{attribute 'qualified_only'}
{attribute 'global_init_slot' := '50500'}
VAR_GLOBAL PERSISTENT
	//These tags are created here because you cannot write directly to local scoped tags(cpt_3144) from outside the POU
	//They are created here then mapped to the local variables in the POU
	//All tags in this GVL MUST have the {attribute 'OPC.UA.DA' :='1'} string above them in order to be exposed to OPC
	//Tags that are ONLY being read from the HMI have their values set in the opc_mapping program
	
		//------------------------------------------------------------------------------------------------------------------

	
	//State Mode
	{attribute 'OPC.UA.DA' :='1'}
	popa_0081_ed_routine_maint : BOOL;
	
//---HMI Commands--------------------------------------------------------------------------------------------------------------------------------------

	//Pumps-----------------------------------------------------------------------------------------------------------------------
	{attribute 'OPC.UA.DA' :='1'}
	popa_0081_u_3112_hmi_start_request: BOOL;
	{attribute 'OPC.UA.DA' :='1'}
	popa_0081_u_3212_hmi_start_request: BOOL;
	{attribute 'OPC.UA.DA' :='1'}
	popa_0081_u_3312_hmi_start_request: BOOL;
	{attribute 'OPC.UA.DA' :='1'}
	popa_0081_u_3160_hmi_start_request: BOOL;
	{attribute 'OPC.UA.DA' :='1'}
	popa_0081_u_3260_hmi_start_request: BOOL;
	{attribute 'OPC.UA.DA' :='1'}
	popa_0081_u_3360_hmi_start_request: BOOL;
	{attribute 'OPC.UA.DA' :='1'}
	popa_0081_u_3370_hmi_start_request: BOOL;
	{attribute 'OPC.UA.DA' :='1'}
	popa_0081_u_3405_hmi_start_request: BOOL;
		
	{attribute 'OPC.UA.DA' :='1'}
	popa_0081_u_3112_hmi_speed_request: REAL;
	{attribute 'OPC.UA.DA' :='1'}
	popa_0081_u_3212_hmi_speed_request: REAL;
	{attribute 'OPC.UA.DA' :='1'}
	popa_0081_u_3312_hmi_speed_request: REAL;
	{attribute 'OPC.UA.DA' :='1'}
	popa_0081_u_3160_hmi_speed_request: REAL;
	{attribute 'OPC.UA.DA' :='1'}
	popa_0081_u_3260_hmi_speed_request: REAL;
	{attribute 'OPC.UA.DA' :='1'}
	popa_0081_u_3360_hmi_speed_request: REAL;
	{attribute 'OPC.UA.DA' :='1'}
	popa_0081_u_3370_hmi_speed_request: REAL;
	{attribute 'OPC.UA.DA' :='1'}
	popa_0081_u_3405_hmi_speed_request: REAL;
	
	//Valves------------------------------------------------------------------------------------------------------------------------------
	{attribute 'OPC.UA.DA' :='1'}
	popa_0081_nv_3110_hmi_open_request: BOOL;
	{attribute 'OPC.UA.DA' :='1'}
	popa_0081_nv_3210_hmi_open_request: BOOL;
	{attribute 'OPC.UA.DA' :='1'}
	popa_0081_nv_3310_hmi_open_request: BOOL;
	{attribute 'OPC.UA.DA' :='1'}
	popa_0081_nv_3135_hmi_open_request: BOOL;
	{attribute 'OPC.UA.DA' :='1'}
	popa_0081_nv_3235_hmi_open_request: BOOL;
	{attribute 'OPC.UA.DA' :='1'}
	popa_0081_nv_3335_hmi_open_request: BOOL;
	{attribute 'OPC.UA.DA' :='1'}
	popa_0081_nv_3372_hmi_open_request: BOOL;
	{attribute 'OPC.UA.DA' :='1'}
	popa_0081_nv_3162_hmi_open_request: BOOL;
	
	//System date time year
	{attribute 'OPC.UA.DA' :='1'}
	popa_0081_system_date_time_year : INT;
	//System date time month
	{attribute 'OPC.UA.DA' :='1'}
	popa_0081_system_date_time_month : INT;
	//System date time day
	{attribute 'OPC.UA.DA' :='1'}
	popa_0081_system_date_time_day : INT;
	//System date time hour
	{attribute 'OPC.UA.DA' :='1'}
	popa_0081_system_date_time_hour : INT;
	//System date time minute
	{attribute 'OPC.UA.DA' :='1'}
	popa_0081_system_date_time_minute : INT;
	//System date time second
	{attribute 'OPC.UA.DA' :='1'}
	popa_0081_system_date_time_second : INT;
	//Hour setpoint for daily reset triggers
	{attribute 'OPC.UA.DA' :='1'}
	popa_0081_daily_reset_hour_setpoint : INT;
	//Minute setpoint for daily reset triggers
	{attribute 'OPC.UA.DA' :='1'}
	popa_0081_daily_reset_minute_setpoint : INT;
	//Alarm acknowledge, acks all alarms, clears lower priority level alarms
	{attribute 'OPC.UA.DA' :='1'}
	popa_0081_alarm_ack : BOOL;
	//Alarm reset, clears higher priority alarms
	{attribute 'OPC.UA.DA' :='1'}
	popa_0081_alarm_reset : BOOL;
	
	
	//------------------------------------------------------------------------------------------------------------------
	//Alarm Priority setpoint
	{attribute 'OPC.UA.DA' :='1'}
	popa_0081_av_3148_position_fail_priority : INT;
	//Alarm delay setpoint(seconds)
	{attribute 'OPC.UA.DA' :='1'}
	popa_0081_av_3148_position_fail_delay_setpoint : INT;
	//Alarm active for HMI
	{attribute 'OPC.UA.DA' :='1'}
	popa_0081_av_3148_position_fail_active : BOOL;
	//Alarm enable
	{attribute 'OPC.UA.DA' :='1'}
	popa_0081_av_3148_position_fail_enable: BOOL;
	//------------------------------------------------------------------------------------------------------------------
	//Alarm Priority setpoint
	{attribute 'OPC.UA.DA' :='1'}
	popa_0081_av_3248_position_fail_priority : INT;
	//Alarm delay setpoint(seconds)
	{attribute 'OPC.UA.DA' :='1'}
	popa_0081_av_3248_position_fail_delay_setpoint : INT;
	//Alarm active for HMI
	{attribute 'OPC.UA.DA' :='1'}
	popa_0081_av_3248_position_fail_active : BOOL;
	//Alarm enable
	{attribute 'OPC.UA.DA' :='1'}
	popa_0081_av_3248_position_fail_enable: BOOL;
	//------------------------------------------------------------------------------------------------------------------
	//Alarm Priority setpoint
	{attribute 'OPC.UA.DA' :='1'}
	popa_0081_av_3348_position_fail_priority : INT;
	//Alarm delay setpoint(seconds)
	{attribute 'OPC.UA.DA' :='1'}
	popa_0081_av_3348_position_fail_delay_setpoint : INT;
	//Alarm active for HMI
	{attribute 'OPC.UA.DA' :='1'}
	popa_0081_av_3348_position_fail_active : BOOL;
	//Alarm enable
	{attribute 'OPC.UA.DA' :='1'}
	popa_0081_av_3348_position_fail_enable: BOOL;
	
	//------------------------------------------------------------------------------------------------------------------
	//Alarm Priority setpoint
	{attribute 'OPC.UA.DA' :='1'}
	popa_0081_nv_3110_fail_to_open_priority : INT;
	//Alarm delay setpoint(seconds)
	{attribute 'OPC.UA.DA' :='1'}
	popa_0081_nv_3110_fail_to_open_delay_setpoint : INT;
	//Alarm active for HMI
	{attribute 'OPC.UA.DA' :='1'}
	popa_0081_nv_3110_fail_to_open_active : BOOL;
	//Alarm enable
	{attribute 'OPC.UA.DA' :='1'}
	popa_0081_nv_3110_fail_to_open_enable: BOOL;
	
	//Alarm Priority setpoint
	{attribute 'OPC.UA.DA' :='1'}
	popa_0081_nv_3110_fail_to_close_priority : INT;
	//Alarm delay setpoint(seconds)
	{attribute 'OPC.UA.DA' :='1'}
	popa_0081_nv_3110_fail_to_close_delay_setpoint : INT;
	//Alarm active for HMI
	{attribute 'OPC.UA.DA' :='1'}
	popa_0081_nv_3110_fail_to_close_active : BOOL;
	//Alarm enable
	{attribute 'OPC.UA.DA' :='1'}
	popa_0081_nv_3110_fail_to_close_enable: BOOL;
	
	//------------------------------------------------------------------------------------------------------------------
	//Alarm Priority setpoint
	{attribute 'OPC.UA.DA' :='1'}
	popa_0081_nv_3210_fail_to_open_priority : INT;
	//Alarm delay setpoint(seconds)
	{attribute 'OPC.UA.DA' :='1'}
	popa_0081_nv_3210_fail_to_open_delay_setpoint : INT;
	//Alarm active for HMI
	{attribute 'OPC.UA.DA' :='1'}
	popa_0081_nv_3210_fail_to_open_active : BOOL;
	//Alarm enable
	{attribute 'OPC.UA.DA' :='1'}
	popa_0081_nv_3210_fail_to_open_enable: BOOL;
	
	//Alarm Priority setpoint
	{attribute 'OPC.UA.DA' :='1'}
	popa_0081_nv_3210_fail_to_close_priority : INT;
	//Alarm delay setpoint(seconds)
	{attribute 'OPC.UA.DA' :='1'}
	popa_0081_nv_3210_fail_to_close_delay_setpoint : INT;
	//Alarm active for HMI
	{attribute 'OPC.UA.DA' :='1'}
	popa_0081_nv_3210_fail_to_close_active : BOOL;
	//Alarm enable
	{attribute 'OPC.UA.DA' :='1'}
	popa_0081_nv_3210_fail_to_close_enable: BOOL;
	
	//------------------------------------------------------------------------------------------------------------------
	//Alarm Priority setpoint
	{attribute 'OPC.UA.DA' :='1'}
	popa_0081_nv_3310_fail_to_open_priority : INT;
	//Alarm delay setpoint(seconds)
	{attribute 'OPC.UA.DA' :='1'}
	popa_0081_nv_3310_fail_to_open_delay_setpoint : INT;
	//Alarm active for HMI
	{attribute 'OPC.UA.DA' :='1'}
	popa_0081_nv_3310_fail_to_open_active : BOOL;
	//Alarm enable
	{attribute 'OPC.UA.DA' :='1'}
	popa_0081_nv_3310_fail_to_open_enable: BOOL;
	
	//Alarm Priority setpoint
	{attribute 'OPC.UA.DA' :='1'}
	popa_0081_nv_3310_fail_to_close_priority : INT;
	//Alarm delay setpoint(seconds)
	{attribute 'OPC.UA.DA' :='1'}
	popa_0081_nv_3310_fail_to_close_delay_setpoint : INT;
	//Alarm active for HMI
	{attribute 'OPC.UA.DA' :='1'}
	popa_0081_nv_3310_fail_to_close_active : BOOL;
	//Alarm enable
	{attribute 'OPC.UA.DA' :='1'}
	popa_0081_nv_3310_fail_to_close_enable: BOOL;
	
	//------------------------------------------------------------------------------------------------------------------
	//Alarm Priority setpoint
	{attribute 'OPC.UA.DA' :='1'}
	popa_0081_nv_3135_fail_to_open_priority : INT;
	//Alarm delay setpoint(seconds)
	{attribute 'OPC.UA.DA' :='1'}
	popa_0081_nv_3135_fail_to_open_delay_setpoint : INT;
	//Alarm active for HMI
	{attribute 'OPC.UA.DA' :='1'}
	popa_0081_nv_3135_fail_to_open_active : BOOL;
	//Alarm enable
	{attribute 'OPC.UA.DA' :='1'}
	popa_0081_nv_3135_fail_to_open_enable: BOOL;
	
	//Alarm Priority setpoint
	{attribute 'OPC.UA.DA' :='1'}
	popa_0081_nv_3135_fail_to_close_priority : INT;
	//Alarm delay setpoint(seconds)
	{attribute 'OPC.UA.DA' :='1'}
	popa_0081_nv_3135_fail_to_close_delay_setpoint : INT;
	//Alarm active for HMI
	{attribute 'OPC.UA.DA' :='1'}
	popa_0081_nv_3135_fail_to_close_active : BOOL;
	//Alarm enable
	{attribute 'OPC.UA.DA' :='1'}
	popa_0081_nv_3135_fail_to_close_enable: BOOL;
	
	//------------------------------------------------------------------------------------------------------------------
	//Alarm Priority setpoint
	{attribute 'OPC.UA.DA' :='1'}
	popa_0081_nv_3235_fail_to_open_priority : INT;
	//Alarm delay setpoint(seconds)
	{attribute 'OPC.UA.DA' :='1'}
	popa_0081_nv_3235_fail_to_open_delay_setpoint : INT;
	//Alarm active for HMI
	{attribute 'OPC.UA.DA' :='1'}
	popa_0081_nv_3235_fail_to_open_active : BOOL;
	//Alarm enable
	{attribute 'OPC.UA.DA' :='1'}
	popa_0081_nv_3235_fail_to_open_enable: BOOL;
	
	//Alarm Priority setpoint
	{attribute 'OPC.UA.DA' :='1'}
	popa_0081_nv_3235_fail_to_close_priority : INT;
	//Alarm delay setpoint(seconds)
	{attribute 'OPC.UA.DA' :='1'}
	popa_0081_nv_3235_fail_to_close_delay_setpoint : INT;
	//Alarm active for HMI
	{attribute 'OPC.UA.DA' :='1'}
	popa_0081_nv_3235_fail_to_close_active : BOOL;
	//Alarm enable
	{attribute 'OPC.UA.DA' :='1'}
	popa_0081_nv_3235_fail_to_close_enable: BOOL;
	
	//------------------------------------------------------------------------------------------------------------------
	//Alarm Priority setpoint
	{attribute 'OPC.UA.DA' :='1'}
	popa_0081_nv_3335_fail_to_open_priority : INT;
	//Alarm delay setpoint(seconds)
	{attribute 'OPC.UA.DA' :='1'}
	popa_0081_nv_3335_fail_to_open_delay_setpoint : INT;
	//Alarm active for HMI
	{attribute 'OPC.UA.DA' :='1'}
	popa_0081_nv_3335_fail_to_open_active : BOOL;
	//Alarm enable
	{attribute 'OPC.UA.DA' :='1'}
	popa_0081_nv_3335_fail_to_open_enable: BOOL;
	
	//Alarm Priority setpoint
	{attribute 'OPC.UA.DA' :='1'}
	popa_0081_nv_3335_fail_to_close_priority : INT;
	//Alarm delay setpoint(seconds)
	{attribute 'OPC.UA.DA' :='1'}
	popa_0081_nv_3335_fail_to_close_delay_setpoint : INT;
	//Alarm active for HMI
	{attribute 'OPC.UA.DA' :='1'}
	popa_0081_nv_3335_fail_to_close_active : BOOL;
	//Alarm enable
	{attribute 'OPC.UA.DA' :='1'}
	popa_0081_nv_3335_fail_to_close_enable: BOOL;
	
	//------------------------------------------------------------------------------------------------------------------
	//Alarm Priority setpoint
	{attribute 'OPC.UA.DA' :='1'}
	popa_0081_nv_3372_fail_to_open_priority : INT;
	//Alarm delay setpoint(seconds)
	{attribute 'OPC.UA.DA' :='1'}
	popa_0081_nv_3372_fail_to_open_delay_setpoint : INT;
	//Alarm active for HMI
	{attribute 'OPC.UA.DA' :='1'}
	popa_0081_nv_3372_fail_to_open_active : BOOL;
	//Alarm enable
	{attribute 'OPC.UA.DA' :='1'}
	popa_0081_nv_3372_fail_to_open_enable: BOOL;
	
	//Alarm Priority setpoint
	{attribute 'OPC.UA.DA' :='1'}
	popa_0081_nv_3372_fail_to_close_priority : INT;
	//Alarm delay setpoint(seconds)
	{attribute 'OPC.UA.DA' :='1'}
	popa_0081_nv_3372_fail_to_close_delay_setpoint : INT;
	//Alarm active for HMI
	{attribute 'OPC.UA.DA' :='1'}
	popa_0081_nv_3372_fail_to_close_active : BOOL;
	//Alarm enable
	{attribute 'OPC.UA.DA' :='1'}
	popa_0081_nv_3372_fail_to_close_enable: BOOL;
	
	//------------------------------------------------------------------------------------------------------------------
	//Alarm Priority setpoint
	{attribute 'OPC.UA.DA' :='1'}
	popa_0081_nv_3162_fail_to_open_priority : INT;
	//Alarm delay setpoint(seconds)
	{attribute 'OPC.UA.DA' :='1'}
	popa_0081_nv_3162_fail_to_open_delay_setpoint : INT;
	//Alarm active for HMI
	{attribute 'OPC.UA.DA' :='1'}
	popa_0081_nv_3162_fail_to_open_active : BOOL;
	//Alarm enable
	{attribute 'OPC.UA.DA' :='1'}
	popa_0081_nv_3162_fail_to_open_enable: BOOL;
	
	//Alarm Priority setpoint
	{attribute 'OPC.UA.DA' :='1'}
	popa_0081_nv_3162_fail_to_close_priority : INT;
	//Alarm delay setpoint(seconds)
	{attribute 'OPC.UA.DA' :='1'}
	popa_0081_nv_3162_fail_to_close_delay_setpoint : INT;
	//Alarm active for HMI
	{attribute 'OPC.UA.DA' :='1'}
	popa_0081_nv_3162_fail_to_close_active : BOOL;
	//Alarm enable
	{attribute 'OPC.UA.DA' :='1'}
	popa_0081_nv_3162_fail_to_close_enable: BOOL;
	


//---Pumps-------------------------------------------------------------------------------------------------------------------------------------
	//------------------------------------------------------------------------------------------------------------------
	//Alarm Priority setpoint
	{attribute 'OPC.UA.DA' :='1'}
	popa_0081_u_3112_fail_to_start_priority : INT;
	//Alarm delay setpoint(seconds)
	{attribute 'OPC.UA.DA' :='1'}
	popa_0081_u_3112_fail_to_start_delay_setpoint : INT;
	//Alarm active for HMI
	{attribute 'OPC.UA.DA' :='1'}
	popa_0081_u_3112_fail_to_start_active : BOOL;
	//Alarm enable
	{attribute 'OPC.UA.DA' :='1'}
	popa_0081_u_3112_fail_to_start_enable: BOOL;
	
	//Alarm Priority setpoint
	{attribute 'OPC.UA.DA' :='1'}
	popa_0081_u_3112_fail_to_stop_priority : INT;
	//Alarm delay setpoint(seconds)
	{attribute 'OPC.UA.DA' :='1'}
	popa_0081_u_3112_fail_to_stop_delay_setpoint : INT;
	//Alarm active for HMI
	{attribute 'OPC.UA.DA' :='1'}
	popa_0081_u_3112_fail_to_stop_active : BOOL;
	//Alarm enable
	{attribute 'OPC.UA.DA' :='1'}
	popa_0081_u_3112_fail_to_stop_enable: BOOL;
	
	//------------------------------------------------------------------------------------------------------------------
	//Alarm Priority setpoint
	{attribute 'OPC.UA.DA' :='1'}
	popa_0081_u_3212_fail_to_start_priority : INT;
	//Alarm delay setpoint(seconds)
	{attribute 'OPC.UA.DA' :='1'}
	popa_0081_u_3212_fail_to_start_delay_setpoint : INT;
	//Alarm active for HMI
	{attribute 'OPC.UA.DA' :='1'}
	popa_0081_u_3212_fail_to_start_active : BOOL;
	//Alarm enable
	{attribute 'OPC.UA.DA' :='1'}
	popa_0081_u_3212_fail_to_start_enable: BOOL;
	
	//Alarm Priority setpoint
	{attribute 'OPC.UA.DA' :='1'}
	popa_0081_u_3212_fail_to_stop_priority : INT;
	//Alarm delay setpoint(seconds)
	{attribute 'OPC.UA.DA' :='1'}
	popa_0081_u_3212_fail_to_stop_delay_setpoint : INT;
	//Alarm active for HMI
	{attribute 'OPC.UA.DA' :='1'}
	popa_0081_u_3212_fail_to_stop_active : BOOL;
	//Alarm enable
	{attribute 'OPC.UA.DA' :='1'}
	popa_0081_u_3212_fail_to_stop_enable: BOOL;
	
	//------------------------------------------------------------------------------------------------------------------
	//Alarm Priority setpoint
	{attribute 'OPC.UA.DA' :='1'}
	popa_0081_u_3312_fail_to_start_priority : INT;
	//Alarm delay setpoint(seconds)
	{attribute 'OPC.UA.DA' :='1'}
	popa_0081_u_3312_fail_to_start_delay_setpoint : INT;
	//Alarm active for HMI
	{attribute 'OPC.UA.DA' :='1'}
	popa_0081_u_3312_fail_to_start_active : BOOL;
	//Alarm enable
	{attribute 'OPC.UA.DA' :='1'}
	popa_0081_u_3312_fail_to_start_enable: BOOL;
	
	//Alarm Priority setpoint
	{attribute 'OPC.UA.DA' :='1'}
	popa_0081_u_3312_fail_to_stop_priority : INT;
	//Alarm delay setpoint(seconds)
	{attribute 'OPC.UA.DA' :='1'}
	popa_0081_u_3312_fail_to_stop_delay_setpoint : INT;
	//Alarm active for HMI
	{attribute 'OPC.UA.DA' :='1'}
	popa_0081_u_3312_fail_to_stop_active : BOOL;
	//Alarm enable
	{attribute 'OPC.UA.DA' :='1'}
	popa_0081_u_3312_fail_to_stop_enable: BOOL;
	
	//------------------------------------------------------------------------------------------------------------------
	//Alarm Priority setpoint
	{attribute 'OPC.UA.DA' :='1'}
	popa_0081_u_3160_fail_to_start_priority : INT;
	//Alarm delay setpoint(seconds)
	{attribute 'OPC.UA.DA' :='1'}
	popa_0081_u_3160_fail_to_start_delay_setpoint : INT;
	//Alarm active for HMI
	{attribute 'OPC.UA.DA' :='1'}
	popa_0081_u_3160_fail_to_start_active : BOOL;
	//Alarm enable
	{attribute 'OPC.UA.DA' :='1'}
	popa_0081_u_3160_fail_to_start_enable: BOOL;
	
	//Alarm Priority setpoint
	{attribute 'OPC.UA.DA' :='1'}
	popa_0081_u_3160_fail_to_stop_priority : INT;
	//Alarm delay setpoint(seconds)
	{attribute 'OPC.UA.DA' :='1'}
	popa_0081_u_3160_fail_to_stop_delay_setpoint : INT;
	//Alarm active for HMI
	{attribute 'OPC.UA.DA' :='1'}
	popa_0081_u_3160_fail_to_stop_active : BOOL;
	//Alarm enable
	{attribute 'OPC.UA.DA' :='1'}
	popa_0081_u_3160_fail_to_stop_enable: BOOL;
	
	//------------------------------------------------------------------------------------------------------------------
	//Alarm Priority setpoint
	{attribute 'OPC.UA.DA' :='1'}
	popa_0081_u_3260_fail_to_start_priority : INT;
	//Alarm delay setpoint(seconds)
	{attribute 'OPC.UA.DA' :='1'}
	popa_0081_u_3260_fail_to_start_delay_setpoint : INT;
	//Alarm active for HMI
	{attribute 'OPC.UA.DA' :='1'}
	popa_0081_u_3260_fail_to_start_active : BOOL;
	//Alarm enable
	{attribute 'OPC.UA.DA' :='1'}
	popa_0081_u_3260_fail_to_start_enable: BOOL;
	
	//Alarm Priority setpoint
	{attribute 'OPC.UA.DA' :='1'}
	popa_0081_u_3260_fail_to_stop_priority : INT;
	//Alarm delay setpoint(seconds)
	{attribute 'OPC.UA.DA' :='1'}
	popa_0081_u_3260_fail_to_stop_delay_setpoint : INT;
	//Alarm active for HMI
	{attribute 'OPC.UA.DA' :='1'}
	popa_0081_u_3260_fail_to_stop_active : BOOL;
	//Alarm enable
	{attribute 'OPC.UA.DA' :='1'}
	popa_0081_u_3260_fail_to_stop_enable: BOOL;
	
	//------------------------------------------------------------------------------------------------------------------
	//Alarm Priority setpoint
	{attribute 'OPC.UA.DA' :='1'}
	popa_0081_u_3360_fail_to_start_priority : INT;
	//Alarm delay setpoint(seconds)
	{attribute 'OPC.UA.DA' :='1'}
	popa_0081_u_3360_fail_to_start_delay_setpoint : INT;
	//Alarm active for HMI
	{attribute 'OPC.UA.DA' :='1'}
	popa_0081_u_3360_fail_to_start_active : BOOL;
	//Alarm enable
	{attribute 'OPC.UA.DA' :='1'}
	popa_0081_u_3360_fail_to_start_enable: BOOL;
	
	//Alarm Priority setpoint
	{attribute 'OPC.UA.DA' :='1'}
	popa_0081_u_3360_fail_to_stop_priority : INT;
	//Alarm delay setpoint(seconds)
	{attribute 'OPC.UA.DA' :='1'}
	popa_0081_u_3360_fail_to_stop_delay_setpoint : INT;
	//Alarm active for HMI
	{attribute 'OPC.UA.DA' :='1'}
	popa_0081_u_3360_fail_to_stop_active : BOOL;
	//Alarm enable
	{attribute 'OPC.UA.DA' :='1'}
	popa_0081_u_3360_fail_to_stop_enable: BOOL;
	
	//------------------------------------------------------------------------------------------------------------------
	//Alarm Priority setpoint
	{attribute 'OPC.UA.DA' :='1'}
	popa_0081_u_3370_fail_to_start_priority : INT;
	//Alarm delay setpoint(seconds)
	{attribute 'OPC.UA.DA' :='1'}
	popa_0081_u_3370_fail_to_start_delay_setpoint : INT;
	//Alarm active for HMI
	{attribute 'OPC.UA.DA' :='1'}
	popa_0081_u_3370_fail_to_start_active : BOOL;
	//Alarm enable
	{attribute 'OPC.UA.DA' :='1'}
	popa_0081_u_3370_fail_to_start_enable: BOOL;
	
	//Alarm Priority setpoint
	{attribute 'OPC.UA.DA' :='1'}
	popa_0081_u_3370_fail_to_stop_priority : INT;
	//Alarm delay setpoint(seconds)
	{attribute 'OPC.UA.DA' :='1'}
	popa_0081_u_3370_fail_to_stop_delay_setpoint : INT;
	//Alarm active for HMI
	{attribute 'OPC.UA.DA' :='1'}
	popa_0081_u_3370_fail_to_stop_active : BOOL;
	//Alarm enable
	{attribute 'OPC.UA.DA' :='1'}
	popa_0081_u_3370_fail_to_stop_enable: BOOL;
	
	//------------------------------------------------------------------------------------------------------------------
	//Alarm Priority setpoint
	{attribute 'OPC.UA.DA' :='1'}
	popa_0081_u_3405_fail_to_start_priority : INT;
	//Alarm delay setpoint(seconds)
	{attribute 'OPC.UA.DA' :='1'}
	popa_0081_u_3405_fail_to_start_delay_setpoint : INT;
	//Alarm active for HMI
	{attribute 'OPC.UA.DA' :='1'}
	popa_0081_u_3405_fail_to_start_active : BOOL;
	//Alarm enable
	{attribute 'OPC.UA.DA' :='1'}
	popa_0081_u_3405_fail_to_start_enable: BOOL;
	
	//Alarm Priority setpoint
	{attribute 'OPC.UA.DA' :='1'}
	popa_0081_u_3405_fail_to_stop_priority : INT;
	//Alarm delay setpoint(seconds)
	{attribute 'OPC.UA.DA' :='1'}
	popa_0081_u_3405_fail_to_stop_delay_setpoint : INT;
	//Alarm active for HMI
	{attribute 'OPC.UA.DA' :='1'}
	popa_0081_u_3405_fail_to_stop_active : BOOL;
	//Alarm enable
	{attribute 'OPC.UA.DA' :='1'}
	popa_0081_u_3405_fail_to_stop_enable: BOOL;

	
	//---------------------------------------------------------------------------------------------------------
	//Raw Min value for analog input
	{attribute 'OPC.UA.DA' :='1'}
	popa_0081_u_3112_speed_command_raw_min : REAL :=0;
	//Raw max value for analog input
	{attribute 'OPC.UA.DA' :='1'}
	popa_0081_u_3112_speed_command_raw_max : REAL :=32767;
	//EU Min value for analog input
	{attribute 'OPC.UA.DA' :='1'}
	popa_0081_u_3112_speed_command_eu_min : REAL;
	//EU Max value for analog input
	{attribute 'OPC.UA.DA' :='1'}
	popa_0081_u_3112_speed_command_eu_max : REAL;
	//Filter factor value for analog input
	{attribute 'OPC.UA.DA' :='1'}
	popa_0081_u_3112_speed_command_filter_factor : REAL;
	//Scaled value for analog input
	{attribute 'OPC.UA.DA' :='1'}
	popa_0081_u_3112_speed_command_scaled_value : REAL;
	
	//Raw Min value for analog input
	{attribute 'OPC.UA.DA' :='1'}
	popa_0081_u_3112_speed_feedback_raw_min : REAL :=0;
	//Raw max value for analog input
	{attribute 'OPC.UA.DA' :='1'}
	popa_0081_u_3112_speed_feedback_raw_max : REAL :=32767;
	//EU Min value for analog input
	{attribute 'OPC.UA.DA' :='1'}
	popa_0081_u_3112_speed_feedback_eu_min : REAL;
	//EU Max value for analog input
	{attribute 'OPC.UA.DA' :='1'}
	popa_0081_u_3112_speed_feedback_eu_max : REAL;
	//Filter factor value for analog input
	{attribute 'OPC.UA.DA' :='1'}
	popa_0081_u_3112_speed_feedback_filter_factor : REAL;
	//Scaled value for analog input
	{attribute 'OPC.UA.DA' :='1'}
	popa_0081_u_3112_speed_feedback_scaled_value : REAL;
	
	
	//---------------------------------------------------------------------------------------------------------
	//Raw Min value for analog input
	{attribute 'OPC.UA.DA' :='1'}
	popa_0081_u_3212_speed_command_raw_min : REAL :=0;
	//Raw max value for analog input
	{attribute 'OPC.UA.DA' :='1'}
	popa_0081_u_3212_speed_command_raw_max : REAL :=32767;
	//EU Min value for analog input
	{attribute 'OPC.UA.DA' :='1'}
	popa_0081_u_3212_speed_command_eu_min : REAL;
	//EU Max value for analog input
	{attribute 'OPC.UA.DA' :='1'}
	popa_0081_u_3212_speed_command_eu_max : REAL;
	//Filter factor value for analog input
	{attribute 'OPC.UA.DA' :='1'}
	popa_0081_u_3212_speed_command_filter_factor : REAL;
	//Scaled value for analog input
	{attribute 'OPC.UA.DA' :='1'}
	popa_0081_u_3212_speed_command_scaled_value : REAL;
	
	//Raw Min value for analog input
	{attribute 'OPC.UA.DA' :='1'}
	popa_0081_u_3212_speed_feedback_raw_min : REAL :=0;
	//Raw max value for analog input
	{attribute 'OPC.UA.DA' :='1'}
	popa_0081_u_3212_speed_feedback_raw_max : REAL :=32767;
	//EU Min value for analog input
	{attribute 'OPC.UA.DA' :='1'}
	popa_0081_u_3212_speed_feedback_eu_min : REAL;
	//EU Max value for analog input
	{attribute 'OPC.UA.DA' :='1'}
	popa_0081_u_3212_speed_feedback_eu_max : REAL;
	//Filter factor value for analog input
	{attribute 'OPC.UA.DA' :='1'}
	popa_0081_u_3212_speed_feedback_filter_factor : REAL;
	//Scaled value for analog input
	{attribute 'OPC.UA.DA' :='1'}
	popa_0081_u_3212_speed_feedback_scaled_value : REAL;
	
	
	//---------------------------------------------------------------------------------------------------------
	//Raw Min value for analog input
	{attribute 'OPC.UA.DA' :='1'}
	popa_0081_u_3312_speed_command_raw_min : REAL :=0;
	//Raw max value for analog input
	{attribute 'OPC.UA.DA' :='1'}
	popa_0081_u_3312_speed_command_raw_max : REAL :=32767;
	//EU Min value for analog input
	{attribute 'OPC.UA.DA' :='1'}
	popa_0081_u_3312_speed_command_eu_min : REAL;
	//EU Max value for analog input
	{attribute 'OPC.UA.DA' :='1'}
	popa_0081_u_3312_speed_command_eu_max : REAL;
	//Filter factor value for analog input
	{attribute 'OPC.UA.DA' :='1'}
	popa_0081_u_3312_speed_command_filter_factor : REAL;
	//Scaled value for analog input
	{attribute 'OPC.UA.DA' :='1'}
	popa_0081_u_3312_speed_command_scaled_value : REAL;
	
	//Raw Min value for analog input
	{attribute 'OPC.UA.DA' :='1'}
	popa_0081_u_3312_speed_feedback_raw_min : REAL :=0;
	//Raw max value for analog input
	{attribute 'OPC.UA.DA' :='1'}
	popa_0081_u_3312_speed_feedback_raw_max : REAL :=32767;
	//EU Min value for analog input
	{attribute 'OPC.UA.DA' :='1'}
	popa_0081_u_3312_speed_feedback_eu_min : REAL;
	//EU Max value for analog input
	{attribute 'OPC.UA.DA' :='1'}
	popa_0081_u_3312_speed_feedback_eu_max : REAL;
	//Filter factor value for analog input
	{attribute 'OPC.UA.DA' :='1'}
	popa_0081_u_3312_speed_feedback_filter_factor : REAL;
	//Scaled value for analog input
	{attribute 'OPC.UA.DA' :='1'}
	popa_0081_u_3312_speed_feedback_scaled_value : REAL;
	
	
	//---------------------------------------------------------------------------------------------------------
	//Raw Min value for analog input
	{attribute 'OPC.UA.DA' :='1'}
	popa_0081_u_3160_speed_command_raw_min : REAL :=0;
	//Raw max value for analog input
	{attribute 'OPC.UA.DA' :='1'}
	popa_0081_u_3160_speed_command_raw_max : REAL :=32767;
	//EU Min value for analog input
	{attribute 'OPC.UA.DA' :='1'}
	popa_0081_u_3160_speed_command_eu_min : REAL;
	//EU Max value for analog input
	{attribute 'OPC.UA.DA' :='1'}
	popa_0081_u_3160_speed_command_eu_max : REAL;
	//Filter factor value for analog input
	{attribute 'OPC.UA.DA' :='1'}
	popa_0081_u_3160_speed_command_filter_factor : REAL;
	//Scaled value for analog input
	{attribute 'OPC.UA.DA' :='1'}
	popa_0081_u_3160_speed_command_scaled_value : REAL;
	
	//Raw Min value for analog input
	{attribute 'OPC.UA.DA' :='1'}
	popa_0081_u_3160_speed_feedback_raw_min : REAL :=0;
	//Raw max value for analog input
	{attribute 'OPC.UA.DA' :='1'}
	popa_0081_u_3160_speed_feedback_raw_max : REAL :=32767;
	//EU Min value for analog input
	{attribute 'OPC.UA.DA' :='1'}
	popa_0081_u_3160_speed_feedback_eu_min : REAL;
	//EU Max value for analog input
	{attribute 'OPC.UA.DA' :='1'}
	popa_0081_u_3160_speed_feedback_eu_max : REAL;
	//Filter factor value for analog input
	{attribute 'OPC.UA.DA' :='1'}
	popa_0081_u_3160_speed_feedback_filter_factor : REAL;
	//Scaled value for analog input
	{attribute 'OPC.UA.DA' :='1'}
	popa_0081_u_3160_speed_feedback_scaled_value : REAL;
	
	
	//---------------------------------------------------------------------------------------------------------
	//Raw Min value for analog input
	{attribute 'OPC.UA.DA' :='1'}
	popa_0081_u_3260_speed_command_raw_min : REAL :=0;
	//Raw max value for analog input
	{attribute 'OPC.UA.DA' :='1'}
	popa_0081_u_3260_speed_command_raw_max : REAL :=32767;
	//EU Min value for analog input
	{attribute 'OPC.UA.DA' :='1'}
	popa_0081_u_3260_speed_command_eu_min : REAL;
	//EU Max value for analog input
	{attribute 'OPC.UA.DA' :='1'}
	popa_0081_u_3260_speed_command_eu_max : REAL;
	//Filter factor value for analog input
	{attribute 'OPC.UA.DA' :='1'}
	popa_0081_u_3260_speed_command_filter_factor : REAL;
	//Scaled value for analog input
	{attribute 'OPC.UA.DA' :='1'}
	popa_0081_u_3260_speed_command_scaled_value : REAL;
	
	//Raw Min value for analog input
	{attribute 'OPC.UA.DA' :='1'}
	popa_0081_u_3260_speed_feedback_raw_min : REAL :=0;
	//Raw max value for analog input
	{attribute 'OPC.UA.DA' :='1'}
	popa_0081_u_3260_speed_feedback_raw_max : REAL :=32767;
	//EU Min value for analog input
	{attribute 'OPC.UA.DA' :='1'}
	popa_0081_u_3260_speed_feedback_eu_min : REAL;
	//EU Max value for analog input
	{attribute 'OPC.UA.DA' :='1'}
	popa_0081_u_3260_speed_feedback_eu_max : REAL;
	//Filter factor value for analog input
	{attribute 'OPC.UA.DA' :='1'}
	popa_0081_u_3260_speed_feedback_filter_factor : REAL;
	//Scaled value for analog input
	{attribute 'OPC.UA.DA' :='1'}
	popa_0081_u_3260_speed_feedback_scaled_value : REAL;
	
	
	//---------------------------------------------------------------------------------------------------------
	//Raw Min value for analog input
	{attribute 'OPC.UA.DA' :='1'}
	popa_0081_u_3360_speed_command_raw_min : REAL :=0;
	//Raw max value for analog input
	{attribute 'OPC.UA.DA' :='1'}
	popa_0081_u_3360_speed_command_raw_max : REAL :=32767;
	//EU Min value for analog input
	{attribute 'OPC.UA.DA' :='1'}
	popa_0081_u_3360_speed_command_eu_min : REAL;
	//EU Max value for analog input
	{attribute 'OPC.UA.DA' :='1'}
	popa_0081_u_3360_speed_command_eu_max : REAL;
	//Filter factor value for analog input
	{attribute 'OPC.UA.DA' :='1'}
	popa_0081_u_3360_speed_command_filter_factor : REAL;
	//Scaled value for analog input
	{attribute 'OPC.UA.DA' :='1'}
	popa_0081_u_3360_speed_command_scaled_value : REAL;
	
	//Raw Min value for analog input
	{attribute 'OPC.UA.DA' :='1'}
	popa_0081_u_3360_speed_feedback_raw_min : REAL :=0;
	//Raw max value for analog input
	{attribute 'OPC.UA.DA' :='1'}
	popa_0081_u_3360_speed_feedback_raw_max : REAL :=32767;
	//EU Min value for analog input
	{attribute 'OPC.UA.DA' :='1'}
	popa_0081_u_3360_speed_feedback_eu_min : REAL;
	//EU Max value for analog input
	{attribute 'OPC.UA.DA' :='1'}
	popa_0081_u_3360_speed_feedback_eu_max : REAL;
	//Filter factor value for analog input
	{attribute 'OPC.UA.DA' :='1'}
	popa_0081_u_3360_speed_feedback_filter_factor : REAL;
	//Scaled value for analog input
	{attribute 'OPC.UA.DA' :='1'}
	popa_0081_u_3360_speed_feedback_scaled_value : REAL;
	
	
	//---------------------------------------------------------------------------------------------------------
	//Raw Min value for analog input
	{attribute 'OPC.UA.DA' :='1'}
	popa_0081_u_3370_speed_command_raw_min : REAL :=0;
	//Raw max value for analog input
	{attribute 'OPC.UA.DA' :='1'}
	popa_0081_u_3370_speed_command_raw_max : REAL :=32767;
	//EU Min value for analog input
	{attribute 'OPC.UA.DA' :='1'}
	popa_0081_u_3370_speed_command_eu_min : REAL;
	//EU Max value for analog input
	{attribute 'OPC.UA.DA' :='1'}
	popa_0081_u_3370_speed_command_eu_max : REAL;
	//Filter factor value for analog input
	{attribute 'OPC.UA.DA' :='1'}
	popa_0081_u_3370_speed_command_filter_factor : REAL;
	//Scaled value for analog input
	{attribute 'OPC.UA.DA' :='1'}
	popa_0081_u_3370_speed_command_scaled_value : REAL;
	
	//Raw Min value for analog input
	{attribute 'OPC.UA.DA' :='1'}
	popa_0081_u_3370_speed_feedback_raw_min : REAL :=0;
	//Raw max value for analog input
	{attribute 'OPC.UA.DA' :='1'}
	popa_0081_u_3370_speed_feedback_raw_max : REAL :=32767;
	//EU Min value for analog input
	{attribute 'OPC.UA.DA' :='1'}
	popa_0081_u_3370_speed_feedback_eu_min : REAL;
	//EU Max value for analog input
	{attribute 'OPC.UA.DA' :='1'}
	popa_0081_u_3370_speed_feedback_eu_max : REAL;
	//Filter factor value for analog input
	{attribute 'OPC.UA.DA' :='1'}
	popa_0081_u_3370_speed_feedback_filter_factor : REAL;
	//Scaled value for analog input
	{attribute 'OPC.UA.DA' :='1'}
	popa_0081_u_3370_speed_feedback_scaled_value : REAL;
	
	
	//---------------------------------------------------------------------------------------------------------
	//Raw Min value for analog input
	{attribute 'OPC.UA.DA' :='1'}
	popa_0081_u_3405_speed_command_raw_min : REAL :=0;
	//Raw max value for analog input
	{attribute 'OPC.UA.DA' :='1'}
	popa_0081_u_3405_speed_command_raw_max : REAL :=32767;
	//EU Min value for analog input
	{attribute 'OPC.UA.DA' :='1'}
	popa_0081_u_3405_speed_command_eu_min : REAL;
	//EU Max value for analog input
	{attribute 'OPC.UA.DA' :='1'}
	popa_0081_u_3405_speed_command_eu_max : REAL;
	//Filter factor value for analog input
	{attribute 'OPC.UA.DA' :='1'}
	popa_0081_u_3405_speed_command_filter_factor : REAL;
	//Scaled value for analog input
	{attribute 'OPC.UA.DA' :='1'}
	popa_0081_u_3405_speed_command_scaled_value : REAL;
	
	//Raw Min value for analog input
	{attribute 'OPC.UA.DA' :='1'}
	popa_0081_u_3405_speed_feedback_raw_min : REAL :=0;
	//Raw max value for analog input
	{attribute 'OPC.UA.DA' :='1'}
	popa_0081_u_3405_speed_feedback_raw_max : REAL :=32767;
	//EU Min value for analog input
	{attribute 'OPC.UA.DA' :='1'}
	popa_0081_u_3405_speed_feedback_eu_min : REAL;
	//EU Max value for analog input
	{attribute 'OPC.UA.DA' :='1'}
	popa_0081_u_3405_speed_feedback_eu_max : REAL;
	//Filter factor value for analog input
	{attribute 'OPC.UA.DA' :='1'}
	popa_0081_u_3405_speed_feedback_filter_factor : REAL;
	//Scaled value for analog input
	{attribute 'OPC.UA.DA' :='1'}
	popa_0081_u_3405_speed_feedback_scaled_value : REAL;
	
//---Valves----------------------------------------------------------------------------------------------------------------------------------------

	//Raw Min value for analog input
	{attribute 'OPC.UA.DA' :='1'}
	popa_0081_av_3148_position_feedback_raw_min : REAL :=0;
	//Raw max value for analog input
	{attribute 'OPC.UA.DA' :='1'}
	popa_0081_av_3148_position_feedback_raw_max : REAL :=32767;
	//EU Min value for analog input
	{attribute 'OPC.UA.DA' :='1'}
	popa_0081_av_3148_position_feedback_eu_min : REAL;
	//EU Max value for analog input
	{attribute 'OPC.UA.DA' :='1'}
	popa_0081_av_3148_position_feedback_eu_max : REAL;
	//Filter factor value for analog input
	{attribute 'OPC.UA.DA' :='1'}
	popa_0081_av_3148_position_feedback_filter_factor : REAL;
	//Scaled value for analog input
	{attribute 'OPC.UA.DA' :='1'}
	popa_0081_av_3148_position_feedback_scaled_value : REAL;
	
	//Raw Min value for analog input
	{attribute 'OPC.UA.DA' :='1'}
	popa_0081_av_3148_position_command_raw_min : REAL :=0;
	//Raw max value for analog input
	{attribute 'OPC.UA.DA' :='1'}
	popa_0081_av_3148_position_command_raw_max : REAL :=32767;
	//EU Min value for analog input
	{attribute 'OPC.UA.DA' :='1'}
	popa_0081_av_3148_position_command_eu_min : REAL;
	//EU Max value for analog input
	{attribute 'OPC.UA.DA' :='1'}
	popa_0081_av_3148_position_command_eu_max : REAL;
	//Filter factor value for analog input
	{attribute 'OPC.UA.DA' :='1'}
	popa_0081_av_3148_position_command_filter_factor : REAL;
	//Scaled value for analog input
	{attribute 'OPC.UA.DA' :='1'}
	popa_0081_av_3148_position_command_scaled_value : REAL;
//-----------------------------------------------------------------------------------------------------------	
	//Raw Min value for analog input
	{attribute 'OPC.UA.DA' :='1'}
	popa_0081_av_3248_position_feedback_raw_min : REAL :=0;
	//Raw max value for analog input
	{attribute 'OPC.UA.DA' :='1'}
	popa_0081_av_3248_position_feedback_raw_max : REAL :=32767;
	//EU Min value for analog input
	{attribute 'OPC.UA.DA' :='1'}
	popa_0081_av_3248_position_feedback_eu_min : REAL;
	//EU Max value for analog input
	{attribute 'OPC.UA.DA' :='1'}
	popa_0081_av_3248_position_feedback_eu_max : REAL;
	//Filter factor value for analog input
	{attribute 'OPC.UA.DA' :='1'}
	popa_0081_av_3248_position_feedback_filter_factor : REAL;
	//Scaled value for analog input
	{attribute 'OPC.UA.DA' :='1'}
	popa_0081_av_3248_position_feedback_scaled_value : REAL;
	
	//Raw Min value for analog input
	{attribute 'OPC.UA.DA' :='1'}
	popa_0081_av_3248_position_command_raw_min : REAL :=0;
	//Raw max value for analog input
	{attribute 'OPC.UA.DA' :='1'}
	popa_0081_av_3248_position_command_raw_max : REAL :=32767;
	//EU Min value for analog input
	{attribute 'OPC.UA.DA' :='1'}
	popa_0081_av_3248_position_command_eu_min : REAL;
	//EU Max value for analog input
	{attribute 'OPC.UA.DA' :='1'}
	popa_0081_av_3248_position_command_eu_max : REAL;
	//Filter factor value for analog input
	{attribute 'OPC.UA.DA' :='1'}
	popa_0081_av_3248_position_command_filter_factor : REAL;
	//Scaled value for analog input
	{attribute 'OPC.UA.DA' :='1'}
	popa_0081_av_3248_position_command_scaled_value : REAL;
//-----------------------------------------------------------------------------------------------------------	

	//Raw Min value for analog input
	{attribute 'OPC.UA.DA' :='1'}
	popa_0081_av_3348_position_feedback_raw_min : REAL :=0;
	//Raw max value for analog input
	{attribute 'OPC.UA.DA' :='1'}
	popa_0081_av_3348_position_feedback_raw_max : REAL :=32767;
	//EU Min value for analog input
	{attribute 'OPC.UA.DA' :='1'}
	popa_0081_av_3348_position_feedback_eu_min : REAL;
	//EU Max value for analog input
	{attribute 'OPC.UA.DA' :='1'}
	popa_0081_av_3348_position_feedback_eu_max : REAL;
	//Filter factor value for analog input
	{attribute 'OPC.UA.DA' :='1'}
	popa_0081_av_3348_position_feedback_filter_factor : REAL;
	//Scaled value for analog input
	{attribute 'OPC.UA.DA' :='1'}
	popa_0081_av_3348_position_feedback_scaled_value : REAL;
	
	//Raw Min value for analog input
	{attribute 'OPC.UA.DA' :='1'}
	popa_0081_av_3348_position_command_raw_min : REAL :=0;
	//Raw max value for analog input
	{attribute 'OPC.UA.DA' :='1'}
	popa_0081_av_3348_position_command_raw_max : REAL :=32767;
	//EU Min value for analog input
	{attribute 'OPC.UA.DA' :='1'}
	popa_0081_av_3348_position_command_eu_min : REAL;
	//EU Max value for analog input
	{attribute 'OPC.UA.DA' :='1'}
	popa_0081_av_3348_position_command_eu_max : REAL;
	//Filter factor value for analog input
	{attribute 'OPC.UA.DA' :='1'}
	popa_0081_av_3348_position_command_filter_factor : REAL;
	//Scaled value for analog input
	{attribute 'OPC.UA.DA' :='1'}
	popa_0081_av_3348_position_command_scaled_value : REAL;
//-----------------------------------------------------------------------------------------------------------		


	//Example motor starter runtime maintenance reset
	{attribute 'OPC.UA.DA' :='1'}
	popa_0081_u_3160_runtime_maint_reset : BOOL;
	//Example motor starter run request
	{attribute 'OPC.UA.DA' :='1'}
	popa_0081_u_3160_run_request : BOOL;
	//Example motor starter runtime today
	{attribute 'OPC.UA.DA' :='1'}
	popa_0081_u_3160_runtime_today : REAL;
	//Example motor starter runtime total
	{attribute 'OPC.UA.DA' :='1'}
	popa_0081_u_3160_runtime_total : REAL;
	//Example motor starter runtime maint
	{attribute 'OPC.UA.DA' :='1'}
	popa_0081_u_3160_runtime_maint : REAL;
	//Example motor starter status, 0=Off, 1=Run, 2=Fault
	{attribute 'OPC.UA.DA' :='1'}
	popa_0081_u_3160_status : REAL;
	
	//--------------------------------------------------------------------------------------------------------------
	//Example motor vfd runtime maintenance reset
	{attribute 'OPC.UA.DA' :='1'}
	popa_0081_u_3112_runtime_maint_reset : BOOL;
	//Example motor vfd run request
	{attribute 'OPC.UA.DA' :='1'}
	popa_0081_u_3112_run_request : BOOL;
	//Example motor vfd speed request
	{attribute 'OPC.UA.DA' :='1'}
	popa_0081_u_3112_speed_request : REAL;
	//Example motor vfd speed feedback
	{attribute 'OPC.UA.DA' :='1'}
	popa_0081_u_3112_speed_feedback : REAL;
	//Example motor vfd runtime today
	{attribute 'OPC.UA.DA' :='1'}
	popa_0081_u_3112_runtime_today : REAL;
	//Example motor vfd runtime total
	{attribute 'OPC.UA.DA' :='1'}
	popa_0081_u_3112_runtime_total : REAL;
	//Example motor vfd runtime maint
	{attribute 'OPC.UA.DA' :='1'}
	popa_0081_u_3112_runtime_maint : REAL;
	//Example motor vfd status, 0=Off, 1=Run, 2=Fault
	{attribute 'OPC.UA.DA' :='1'}
	popa_0081_u_3112_status : REAL;
	
	//--------------------------------------------------------------------------------------------------------------
	//Example motor vfd runtime maintenance reset
	{attribute 'OPC.UA.DA' :='1'}
	popa_0081_u_3212_runtime_maint_reset : BOOL;
	//Example motor vfd run request
	{attribute 'OPC.UA.DA' :='1'}
	popa_0081_u_3212_run_request : BOOL;
	//Example motor vfd speed request
	{attribute 'OPC.UA.DA' :='1'}
	popa_0081_u_3212_speed_request : REAL;
	//Example motor vfd speed feedback
	{attribute 'OPC.UA.DA' :='1'}
	popa_0081_u_3212_speed_feedback : REAL;
	//Example motor vfd runtime today
	{attribute 'OPC.UA.DA' :='1'}
	popa_0081_u_3212_runtime_today : REAL;
	//Example motor vfd runtime total
	{attribute 'OPC.UA.DA' :='1'}
	popa_0081_u_3212_runtime_total : REAL;
	//Example motor vfd runtime maint
	{attribute 'OPC.UA.DA' :='1'}
	popa_0081_u_3212_runtime_maint : REAL;
	//Example motor vfd status, 0=Off, 1=Run, 2=Fault
	{attribute 'OPC.UA.DA' :='1'}
	popa_0081_u_3212_status : REAL;
	
	//--------------------------------------------------------------------------------------------------------------
	//Example motor vfd runtime maintenance reset
	{attribute 'OPC.UA.DA' :='1'}
	popa_0081_u_3312_runtime_maint_reset : BOOL;
	//Example motor vfd run request
	{attribute 'OPC.UA.DA' :='1'}
	popa_0081_u_3312_run_request : BOOL;
	//Example motor vfd speed request
	{attribute 'OPC.UA.DA' :='1'}
	popa_0081_u_3312_speed_request : REAL;
	//Example motor vfd speed feedback
	{attribute 'OPC.UA.DA' :='1'}
	popa_0081_u_3312_speed_feedback : REAL;
	//Example motor vfd runtime today
	{attribute 'OPC.UA.DA' :='1'}
	popa_0081_u_3312_runtime_today : REAL;
	//Example motor vfd runtime total
	{attribute 'OPC.UA.DA' :='1'}
	popa_0081_u_3312_runtime_total : REAL;
	//Example motor vfd runtime maint
	{attribute 'OPC.UA.DA' :='1'}
	popa_0081_u_3312_runtime_maint : REAL;
	//Example motor vfd status, 0=Off, 1=Run, 2=Fault
	{attribute 'OPC.UA.DA' :='1'}
	popa_0081_u_3312_status : REAL;
	
	//--------------------------------------------------------------------------------------------------------------
	
	//Example motor vfd speed request
	{attribute 'OPC.UA.DA' :='1'}
	popa_0081_u_3160_speed_request : REAL;
	//Example motor vfd speed feedback
	{attribute 'OPC.UA.DA' :='1'}
	popa_0081_u_3160_speed_feedback : REAL;

	
	
	//--------------------------------------------------------------------------------------------------------------
	//Example motor vfd runtime maintenance reset
	{attribute 'OPC.UA.DA' :='1'}
	popa_0081_u_3260_runtime_maint_reset : BOOL;
	//Example motor vfd run request
	{attribute 'OPC.UA.DA' :='1'}
	popa_0081_u_3260_run_request : BOOL;
	//Example motor vfd speed request
	{attribute 'OPC.UA.DA' :='1'}
	popa_0081_u_3260_speed_request : REAL;
	//Example motor vfd speed feedback
	{attribute 'OPC.UA.DA' :='1'}
	popa_0081_u_3260_speed_feedback : REAL;
	//Example motor vfd runtime today
	{attribute 'OPC.UA.DA' :='1'}
	popa_0081_u_3260_runtime_today : REAL;
	//Example motor vfd runtime total
	{attribute 'OPC.UA.DA' :='1'}
	popa_0081_u_3260_runtime_total : REAL;
	//Example motor vfd runtime maint
	{attribute 'OPC.UA.DA' :='1'}
	popa_0081_u_3260_runtime_maint : REAL;
	//Example motor vfd status, 0=Off, 1=Run, 2=Fault
	{attribute 'OPC.UA.DA' :='1'}
	popa_0081_u_3260_status : REAL;
	
	//--------------------------------------------------------------------------------------------------------------
	//Example motor vfd runtime maintenance reset
	{attribute 'OPC.UA.DA' :='1'}
	popa_0081_u_3360_runtime_maint_reset : BOOL;
	//Example motor vfd run request
	{attribute 'OPC.UA.DA' :='1'}
	popa_0081_u_3360_run_request : BOOL;
	//Example motor vfd speed request
	{attribute 'OPC.UA.DA' :='1'}
	popa_0081_u_3360_speed_request : REAL;
	//Example motor vfd speed feedback
	{attribute 'OPC.UA.DA' :='1'}
	popa_0081_u_3360_speed_feedback : REAL;
	//Example motor vfd runtime today
	{attribute 'OPC.UA.DA' :='1'}
	popa_0081_u_3360_runtime_today : REAL;
	//Example motor vfd runtime total
	{attribute 'OPC.UA.DA' :='1'}
	popa_0081_u_3360_runtime_total : REAL;
	//Example motor vfd runtime maint
	{attribute 'OPC.UA.DA' :='1'}
	popa_0081_u_3360_runtime_maint : REAL;
	//Example motor vfd status, 0=Off, 1=Run, 2=Fault
	{attribute 'OPC.UA.DA' :='1'}
	popa_0081_u_3360_status : REAL;
	
	//--------------------------------------------------------------------------------------------------------------
	//Example motor vfd runtime maintenance reset
	{attribute 'OPC.UA.DA' :='1'}
	popa_0081_u_3370_runtime_maint_reset : BOOL;
	//Example motor vfd run request
	{attribute 'OPC.UA.DA' :='1'}
	popa_0081_u_3370_run_request : BOOL;
	//Example motor vfd speed request
	{attribute 'OPC.UA.DA' :='1'}
	popa_0081_u_3370_speed_request : REAL;
	//Example motor vfd speed feedback
	{attribute 'OPC.UA.DA' :='1'}
	popa_0081_u_3370_speed_feedback : REAL;
	//Example motor vfd runtime today
	{attribute 'OPC.UA.DA' :='1'}
	popa_0081_u_3370_runtime_today : REAL;
	//Example motor vfd runtime total
	{attribute 'OPC.UA.DA' :='1'}
	popa_0081_u_3370_runtime_total : REAL;
	//Example motor vfd runtime maint
	{attribute 'OPC.UA.DA' :='1'}
	popa_0081_u_3370_runtime_maint : REAL;
	//Example motor vfd status, 0=Off, 1=Run, 2=Fault
	{attribute 'OPC.UA.DA' :='1'}
	popa_0081_u_3370_status : REAL;
	
	//--------------------------------------------------------------------------------------------------------------
	//Example motor vfd runtime maintenance reset
	{attribute 'OPC.UA.DA' :='1'}
	popa_0081_u_3405_runtime_maint_reset : BOOL;
	//Example motor vfd run request
	{attribute 'OPC.UA.DA' :='1'}
	popa_0081_u_3405_run_request : BOOL;
	//Example motor vfd speed request
	{attribute 'OPC.UA.DA' :='1'}
	popa_0081_u_3405_speed_request : REAL;
	//Example motor vfd speed feedback
	{attribute 'OPC.UA.DA' :='1'}
	popa_0081_u_3405_speed_feedback : REAL;
	//Example motor vfd runtime today
	{attribute 'OPC.UA.DA' :='1'}
	popa_0081_u_3405_runtime_today : REAL;
	//Example motor vfd runtime total
	{attribute 'OPC.UA.DA' :='1'}
	popa_0081_u_3405_runtime_total : REAL;
	//Example motor vfd runtime maint
	{attribute 'OPC.UA.DA' :='1'}
	popa_0081_u_3405_runtime_maint : REAL;
	//Example motor vfd status, 0=Off, 1=Run, 2=Fault
	{attribute 'OPC.UA.DA' :='1'}
	popa_0081_u_3405_status : REAL;
	
	
	//Analog valve position request
	{attribute 'OPC.UA.DA' :='1'}
	popa_0081_av_3148_position_feedback : REAL;
	//Example analog valve position request
	{attribute 'OPC.UA.DA' :='1'}
	popa_0081_av_3148_position_request : REAL;
	//Example analog valve position fail deadband
	{attribute 'OPC.UA.DA' :='1'}
	popa_0081_av_3148_position_deadband_sp : REAL;
	//Example analog valve position requested when in fault state
	{attribute 'OPC.UA.DA' :='1'}
	popa_0081_av_3148_position_faulted : REAL;
	//Example analog valve status
	{attribute 'OPC.UA.DA' :='1'}
	popa_0081_av_3148_status : INT;
	//-------------------------------------------------------------------------------------------
		{attribute 'OPC.UA.DA' :='1'}
	popa_0081_av_3248_position_feedback : REAL;
	//Example analog valve position request
	{attribute 'OPC.UA.DA' :='1'}
	popa_0081_av_3248_position_request : REAL;
	//Example analog valve position fail deadband
	{attribute 'OPC.UA.DA' :='1'}
	popa_0081_av_3248_position_deadband_sp : REAL;
	//Example analog valve position requested when in fault state
	{attribute 'OPC.UA.DA' :='1'}
	popa_0081_av_3248_position_faulted : REAL;
	//Example analog valve status
	{attribute 'OPC.UA.DA' :='1'}
	popa_0081_av_3248_status : INT;
	//-------------------------------------------------------------------------------------------
		{attribute 'OPC.UA.DA' :='1'}
	popa_0081_av_3348_position_feedback : REAL;
	//Example analog valve position request
	{attribute 'OPC.UA.DA' :='1'}
	popa_0081_av_3348_position_request : REAL;
	//Example analog valve position fail deadband
	{attribute 'OPC.UA.DA' :='1'}
	popa_0081_av_3348_position_deadband_sp : REAL;
	//Example analog valve position requested when in fault state
	{attribute 'OPC.UA.DA' :='1'}
	popa_0081_av_3348_position_faulted : REAL;
	//Example analog valve status
	{attribute 'OPC.UA.DA' :='1'}
	popa_0081_av_3348_status : INT;
	//-------------------------------------------------------------------------------------------
	//Example digital valve open request
	{attribute 'OPC.UA.DA' :='1'}
	popa_0081_nv_3372_open_request : BOOL;
	//Example digital valve status
	{attribute 'OPC.UA.DA' :='1'}
	popa_0081_nv_3372_status : INT;
	
//---Sensors----------------------------------------------------------------------------------------------------------------------------	
	//---cpt_3144-----------------------------------------------------------------------------------------------------------------------
	//Alarm Priority setpoint
	{attribute 'OPC.UA.DA' :='1'}
	popa_0081_cpt_3144_low_low_priority : INT;
	//Alarm delay setpoint(seconds)
	{attribute 'OPC.UA.DA' :='1'}
	popa_0081_cpt_3144_low_low_delay_setpoint : INT;
	//Alarm active for HMI
	{attribute 'OPC.UA.DA' :='1'}
	popa_0081_cpt_3144_low_low_active : BOOL;
	//Analog Alarm Setpoint
	{attribute 'OPC.UA.DA' :='1'}
	popa_0081_cpt_3144_low_low_setpoint : REAL;
	//Alarm enable
	{attribute 'OPC.UA.DA' :='1'}
	popa_0081_cpt_3144_low_low_enable: BOOL;
	
	//Alarm Priority setpoint
	{attribute 'OPC.UA.DA' :='1'}
	popa_0081_cpt_3144_low_priority : INT;
	//Alarm delay setpoint(seconds)
	{attribute 'OPC.UA.DA' :='1'}
	popa_0081_cpt_3144_low_delay_setpoint : INT;
	//Alarm active for HMI
	{attribute 'OPC.UA.DA' :='1'}
	popa_0081_cpt_3144_low_active : BOOL;
	//Analog Alarm Setpoint
	{attribute 'OPC.UA.DA' :='1'}
	popa_0081_cpt_3144_low_setpoint : REAL;
	//Alarm enable
	{attribute 'OPC.UA.DA' :='1'}
	popa_0081_cpt_3144_low_enable: BOOL;
	
	//Alarm Priority setpoint
	{attribute 'OPC.UA.DA' :='1'}
	popa_0081_cpt_3144_high_priority : INT;
	//Alarm delay setpoint(seconds)
	{attribute 'OPC.UA.DA' :='1'}
	popa_0081_cpt_3144_high_delay_setpoint : INT;
	//Alarm active for HMI
	{attribute 'OPC.UA.DA' :='1'}
	popa_0081_cpt_3144_high_active : BOOL;
	//Analog Alarm Setpoint
	{attribute 'OPC.UA.DA' :='1'}
	popa_0081_cpt_3144_high_setpoint : REAL;
	//Alarm enable
	{attribute 'OPC.UA.DA' :='1'}
	popa_0081_cpt_3144_high_enable: BOOL;
	
	//Alarm Priority setpoint
	{attribute 'OPC.UA.DA' :='1'}
	popa_0081_cpt_3144_high_high_priority : INT;
	//Alarm delay setpoint(seconds)
	{attribute 'OPC.UA.DA' :='1'}
	popa_0081_cpt_3144_high_high_delay_setpoint : INT;
	//Alarm active for HMI
	{attribute 'OPC.UA.DA' :='1'}
	popa_0081_cpt_3144_high_high_active : BOOL;
	//Analog Alarm Setpoint
	{attribute 'OPC.UA.DA' :='1'}
	popa_0081_cpt_3144_high_high_setpoint : REAL;
	//Alarm enable
	{attribute 'OPC.UA.DA' :='1'}
	popa_0081_cpt_3144_high_high_enable: BOOL;
	
	
	//Raw Min value for analog input
	{attribute 'OPC.UA.DA' :='1'}
	popa_0081_cpt_3144_raw_min : REAL :=0;
	//Raw max value for analog input
	{attribute 'OPC.UA.DA' :='1'}
	popa_0081_cpt_3144_raw_max : REAL :=32767;
	//EU Min value for analog input
	{attribute 'OPC.UA.DA' :='1'}
	popa_0081_cpt_3144_eu_min : REAL;
	//EU Max value for analog input
	{attribute 'OPC.UA.DA' :='1'}
	popa_0081_cpt_3144_eu_max : REAL;
	//Filter factor value for analog input
	{attribute 'OPC.UA.DA' :='1'}
	popa_0081_cpt_3144_filter_factor : REAL;
	//Scaled value for analog input
	{attribute 'OPC.UA.DA' :='1'}
	popa_0081_cpt_3144_scaled_value : REAL;

	//---pt_3119-----------------------------------------------------------------------------------------------------------------------
	//Alarm Priority setpoint
	{attribute 'OPC.UA.DA' :='1'}
	popa_0081_pt_3119_low_low_priority : INT;
	//Alarm delay setpoint(seconds)
	{attribute 'OPC.UA.DA' :='1'}
	popa_0081_pt_3119_low_low_delay_setpoint : INT;
	//Alarm active for HMI
	{attribute 'OPC.UA.DA' :='1'}
	popa_0081_pt_3119_low_low_active : BOOL;
	//Analog Alarm Setpoint
	{attribute 'OPC.UA.DA' :='1'}
	popa_0081_pt_3119_low_low_setpoint : REAL;
	//Alarm enable
	{attribute 'OPC.UA.DA' :='1'}
	popa_0081_pt_3119_low_low_enable: BOOL;
	
	//Alarm Priority setpoint
	{attribute 'OPC.UA.DA' :='1'}
	popa_0081_pt_3119_low_priority : INT;
	//Alarm delay setpoint(seconds)
	{attribute 'OPC.UA.DA' :='1'}
	popa_0081_pt_3119_low_delay_setpoint : INT;
	//Alarm active for HMI
	{attribute 'OPC.UA.DA' :='1'}
	popa_0081_pt_3119_low_active : BOOL;
	//Analog Alarm Setpoint
	{attribute 'OPC.UA.DA' :='1'}
	popa_0081_pt_3119_low_setpoint : REAL;
	//Alarm enable
	{attribute 'OPC.UA.DA' :='1'}
	popa_0081_pt_3119_low_enable: BOOL;
	
	//Alarm Priority setpoint
	{attribute 'OPC.UA.DA' :='1'}
	popa_0081_pt_3119_high_priority : INT;
	//Alarm delay setpoint(seconds)
	{attribute 'OPC.UA.DA' :='1'}
	popa_0081_pt_3119_high_delay_setpoint : INT;
	//Alarm active for HMI
	{attribute 'OPC.UA.DA' :='1'}
	popa_0081_pt_3119_high_active : BOOL;
	//Analog Alarm Setpoint
	{attribute 'OPC.UA.DA' :='1'}
	popa_0081_pt_3119_high_setpoint : REAL;
	//Alarm enable
	{attribute 'OPC.UA.DA' :='1'}
	popa_0081_pt_3119_high_enable: BOOL;
	
	//Alarm Priority setpoint
	{attribute 'OPC.UA.DA' :='1'}
	popa_0081_pt_3119_high_high_priority : INT;
	//Alarm delay setpoint(seconds)
	{attribute 'OPC.UA.DA' :='1'}
	popa_0081_pt_3119_high_high_delay_setpoint : INT;
	//Alarm active for HMI
	{attribute 'OPC.UA.DA' :='1'}
	popa_0081_pt_3119_high_high_active : BOOL;
	//Analog Alarm Setpoint
	{attribute 'OPC.UA.DA' :='1'}
	popa_0081_pt_3119_high_high_setpoint : REAL;
	//Alarm enable
	{attribute 'OPC.UA.DA' :='1'}
	popa_0081_pt_3119_high_high_enable: BOOL;
	
	
	//Raw Min value for analog input
	{attribute 'OPC.UA.DA' :='1'}
	popa_0081_pt_3119_raw_min : REAL :=0;
	//Raw max value for analog input
	{attribute 'OPC.UA.DA' :='1'}
	popa_0081_pt_3119_raw_max : REAL :=32767;
	//EU Min value for analog input
	{attribute 'OPC.UA.DA' :='1'}
	popa_0081_pt_3119_eu_min : REAL;
	//EU Max value for analog input
	{attribute 'OPC.UA.DA' :='1'}
	popa_0081_pt_3119_eu_max : REAL;
	//Filter factor value for analog input
	{attribute 'OPC.UA.DA' :='1'}
	popa_0081_pt_3119_filter_factor : REAL;
	//Scaled value for analog input
	{attribute 'OPC.UA.DA' :='1'}
	popa_0081_pt_3119_scaled_value : REAL;
	
	//---pt_3219-----------------------------------------------------------------------------------------------------------------------
	//Alarm Priority setpoint
	{attribute 'OPC.UA.DA' :='1'}
	popa_0081_pt_3219_low_low_priority : INT;
	//Alarm delay setpoint(seconds)
	{attribute 'OPC.UA.DA' :='1'}
	popa_0081_pt_3219_low_low_delay_setpoint : INT;
	//Alarm active for HMI
	{attribute 'OPC.UA.DA' :='1'}
	popa_0081_pt_3219_low_low_active : BOOL;
	//Analog Alarm Setpoint
	{attribute 'OPC.UA.DA' :='1'}
	popa_0081_pt_3219_low_low_setpoint : REAL;
	//Alarm enable
	{attribute 'OPC.UA.DA' :='1'}
	popa_0081_pt_3219_low_low_enable: BOOL;
	
	//Alarm Priority setpoint
	{attribute 'OPC.UA.DA' :='1'}
	popa_0081_pt_3219_low_priority : INT;
	//Alarm delay setpoint(seconds)
	{attribute 'OPC.UA.DA' :='1'}
	popa_0081_pt_3219_low_delay_setpoint : INT;
	//Alarm active for HMI
	{attribute 'OPC.UA.DA' :='1'}
	popa_0081_pt_3219_low_active : BOOL;
	//Analog Alarm Setpoint
	{attribute 'OPC.UA.DA' :='1'}
	popa_0081_pt_3219_low_setpoint : REAL;
	//Alarm enable
	{attribute 'OPC.UA.DA' :='1'}
	popa_0081_pt_3219_low_enable: BOOL;
	
	//Alarm Priority setpoint
	{attribute 'OPC.UA.DA' :='1'}
	popa_0081_pt_3219_high_priority : INT;
	//Alarm delay setpoint(seconds)
	{attribute 'OPC.UA.DA' :='1'}
	popa_0081_pt_3219_high_delay_setpoint : INT;
	//Alarm active for HMI
	{attribute 'OPC.UA.DA' :='1'}
	popa_0081_pt_3219_high_active : BOOL;
	//Analog Alarm Setpoint
	{attribute 'OPC.UA.DA' :='1'}
	popa_0081_pt_3219_high_setpoint : REAL;
	//Alarm enable
	{attribute 'OPC.UA.DA' :='1'}
	popa_0081_pt_3219_high_enable: BOOL;
	
	//Alarm Priority setpoint
	{attribute 'OPC.UA.DA' :='1'}
	popa_0081_pt_3219_high_high_priority : INT;
	//Alarm delay setpoint(seconds)
	{attribute 'OPC.UA.DA' :='1'}
	popa_0081_pt_3219_high_high_delay_setpoint : INT;
	//Alarm active for HMI
	{attribute 'OPC.UA.DA' :='1'}
	popa_0081_pt_3219_high_high_active : BOOL;
	//Analog Alarm Setpoint
	{attribute 'OPC.UA.DA' :='1'}
	popa_0081_pt_3219_high_high_setpoint : REAL;
	//Alarm enable
	{attribute 'OPC.UA.DA' :='1'}
	popa_0081_pt_3219_high_high_enable: BOOL;
	
	
	//Raw Min value for analog input
	{attribute 'OPC.UA.DA' :='1'}
	popa_0081_pt_3219_raw_min : REAL :=0;
	//Raw max value for analog input
	{attribute 'OPC.UA.DA' :='1'}
	popa_0081_pt_3219_raw_max : REAL :=32767;
	//EU Min value for analog input
	{attribute 'OPC.UA.DA' :='1'}
	popa_0081_pt_3219_eu_min : REAL;
	//EU Max value for analog input
	{attribute 'OPC.UA.DA' :='1'}
	popa_0081_pt_3219_eu_max : REAL;
	//Filter factor value for analog input
	{attribute 'OPC.UA.DA' :='1'}
	popa_0081_pt_3219_filter_factor : REAL;
	//Scaled value for analog input
	{attribute 'OPC.UA.DA' :='1'}
	popa_0081_pt_3219_scaled_value : REAL;
	
	//---pt_3319-----------------------------------------------------------------------------------------------------------------------
	//Alarm Priority setpoint
	{attribute 'OPC.UA.DA' :='1'}
	popa_0081_pt_3319_low_low_priority : INT;
	//Alarm delay setpoint(seconds)
	{attribute 'OPC.UA.DA' :='1'}
	popa_0081_pt_3319_low_low_delay_setpoint : INT;
	//Alarm active for HMI
	{attribute 'OPC.UA.DA' :='1'}
	popa_0081_pt_3319_low_low_active : BOOL;
	//Analog Alarm Setpoint
	{attribute 'OPC.UA.DA' :='1'}
	popa_0081_pt_3319_low_low_setpoint : REAL;
	//Alarm enable
	{attribute 'OPC.UA.DA' :='1'}
	popa_0081_pt_3319_low_low_enable: BOOL;
	
	//Alarm Priority setpoint
	{attribute 'OPC.UA.DA' :='1'}
	popa_0081_pt_3319_low_priority : INT;
	//Alarm delay setpoint(seconds)
	{attribute 'OPC.UA.DA' :='1'}
	popa_0081_pt_3319_low_delay_setpoint : INT;
	//Alarm active for HMI
	{attribute 'OPC.UA.DA' :='1'}
	popa_0081_pt_3319_low_active : BOOL;
	//Analog Alarm Setpoint
	{attribute 'OPC.UA.DA' :='1'}
	popa_0081_pt_3319_low_setpoint : REAL;
	//Alarm enable
	{attribute 'OPC.UA.DA' :='1'}
	popa_0081_pt_3319_low_enable: BOOL;
	
	//Alarm Priority setpoint
	{attribute 'OPC.UA.DA' :='1'}
	popa_0081_pt_3319_high_priority : INT;
	//Alarm delay setpoint(seconds)
	{attribute 'OPC.UA.DA' :='1'}
	popa_0081_pt_3319_high_delay_setpoint : INT;
	//Alarm active for HMI
	{attribute 'OPC.UA.DA' :='1'}
	popa_0081_pt_3319_high_active : BOOL;
	//Analog Alarm Setpoint
	{attribute 'OPC.UA.DA' :='1'}
	popa_0081_pt_3319_high_setpoint : REAL;
	//Alarm enable
	{attribute 'OPC.UA.DA' :='1'}
	popa_0081_pt_3319_high_enable: BOOL;
	
	//Alarm Priority setpoint
	{attribute 'OPC.UA.DA' :='1'}
	popa_0081_pt_3319_high_high_priority : INT;
	//Alarm delay setpoint(seconds)
	{attribute 'OPC.UA.DA' :='1'}
	popa_0081_pt_3319_high_high_delay_setpoint : INT;
	//Alarm active for HMI
	{attribute 'OPC.UA.DA' :='1'}
	popa_0081_pt_3319_high_high_active : BOOL;
	//Analog Alarm Setpoint
	{attribute 'OPC.UA.DA' :='1'}
	popa_0081_pt_3319_high_high_setpoint : REAL;
	//Alarm enable
	{attribute 'OPC.UA.DA' :='1'}
	popa_0081_pt_3319_high_high_enable: BOOL;
	
	
	//Raw Min value for analog input
	{attribute 'OPC.UA.DA' :='1'}
	popa_0081_pt_3319_raw_min : REAL :=0;
	//Raw max value for analog input
	{attribute 'OPC.UA.DA' :='1'}
	popa_0081_pt_3319_raw_max : REAL :=32767;
	//EU Min value for analog input
	{attribute 'OPC.UA.DA' :='1'}
	popa_0081_pt_3319_eu_min : REAL;
	//EU Max value for analog input
	{attribute 'OPC.UA.DA' :='1'}
	popa_0081_pt_3319_eu_max : REAL;
	//Filter factor value for analog input
	{attribute 'OPC.UA.DA' :='1'}
	popa_0081_pt_3319_filter_factor : REAL;
	//Scaled value for analog input
	{attribute 'OPC.UA.DA' :='1'}
	popa_0081_pt_3319_scaled_value : REAL;
	
	//---pt_3141-----------------------------------------------------------------------------------------------------------------------
	//Alarm Priority setpoint
	{attribute 'OPC.UA.DA' :='1'}
	popa_0081_pt_3141_low_low_priority : INT;
	//Alarm delay setpoint(seconds)
	{attribute 'OPC.UA.DA' :='1'}
	popa_0081_pt_3141_low_low_delay_setpoint : INT;
	//Alarm active for HMI
	{attribute 'OPC.UA.DA' :='1'}
	popa_0081_pt_3141_low_low_active : BOOL;
	//Analog Alarm Setpoint
	{attribute 'OPC.UA.DA' :='1'}
	popa_0081_pt_3141_low_low_setpoint : REAL;
	//Alarm enable
	{attribute 'OPC.UA.DA' :='1'}
	popa_0081_pt_3141_low_low_enable: BOOL;
	
	//Alarm Priority setpoint
	{attribute 'OPC.UA.DA' :='1'}
	popa_0081_pt_3141_low_priority : INT;
	//Alarm delay setpoint(seconds)
	{attribute 'OPC.UA.DA' :='1'}
	popa_0081_pt_3141_low_delay_setpoint : INT;
	//Alarm active for HMI
	{attribute 'OPC.UA.DA' :='1'}
	popa_0081_pt_3141_low_active : BOOL;
	//Analog Alarm Setpoint
	{attribute 'OPC.UA.DA' :='1'}
	popa_0081_pt_3141_low_setpoint : REAL;
	//Alarm enable
	{attribute 'OPC.UA.DA' :='1'}
	popa_0081_pt_3141_low_enable: BOOL;
	
	//Alarm Priority setpoint
	{attribute 'OPC.UA.DA' :='1'}
	popa_0081_pt_3141_high_priority : INT;
	//Alarm delay setpoint(seconds)
	{attribute 'OPC.UA.DA' :='1'}
	popa_0081_pt_3141_high_delay_setpoint : INT;
	//Alarm active for HMI
	{attribute 'OPC.UA.DA' :='1'}
	popa_0081_pt_3141_high_active : BOOL;
	//Analog Alarm Setpoint
	{attribute 'OPC.UA.DA' :='1'}
	popa_0081_pt_3141_high_setpoint : REAL;
	//Alarm enable
	{attribute 'OPC.UA.DA' :='1'}
	popa_0081_pt_3141_high_enable: BOOL;
	
	//Alarm Priority setpoint
	{attribute 'OPC.UA.DA' :='1'}
	popa_0081_pt_3141_high_high_priority : INT;
	//Alarm delay setpoint(seconds)
	{attribute 'OPC.UA.DA' :='1'}
	popa_0081_pt_3141_high_high_delay_setpoint : INT;
	//Alarm active for HMI
	{attribute 'OPC.UA.DA' :='1'}
	popa_0081_pt_3141_high_high_active : BOOL;
	//Analog Alarm Setpoint
	{attribute 'OPC.UA.DA' :='1'}
	popa_0081_pt_3141_high_high_setpoint : REAL;
	//Alarm enable
	{attribute 'OPC.UA.DA' :='1'}
	popa_0081_pt_3141_high_high_enable: BOOL;
	
	
	//Raw Min value for analog input
	{attribute 'OPC.UA.DA' :='1'}
	popa_0081_pt_3141_raw_min : REAL :=0;
	//Raw max value for analog input
	{attribute 'OPC.UA.DA' :='1'}
	popa_0081_pt_3141_raw_max : REAL :=32767;
	//EU Min value for analog input
	{attribute 'OPC.UA.DA' :='1'}
	popa_0081_pt_3141_eu_min : REAL;
	//EU Max value for analog input
	{attribute 'OPC.UA.DA' :='1'}
	popa_0081_pt_3141_eu_max : REAL;
	//Filter factor value for analog input
	{attribute 'OPC.UA.DA' :='1'}
	popa_0081_pt_3141_filter_factor : REAL;
	//Scaled value for analog input
	{attribute 'OPC.UA.DA' :='1'}
	popa_0081_pt_3141_scaled_value : REAL;
	
	//---pt_3241-----------------------------------------------------------------------------------------------------------------------
	//Alarm Priority setpoint
	{attribute 'OPC.UA.DA' :='1'}
	popa_0081_pt_3241_low_low_priority : INT;
	//Alarm delay setpoint(seconds)
	{attribute 'OPC.UA.DA' :='1'}
	popa_0081_pt_3241_low_low_delay_setpoint : INT;
	//Alarm active for HMI
	{attribute 'OPC.UA.DA' :='1'}
	popa_0081_pt_3241_low_low_active : BOOL;
	//Analog Alarm Setpoint
	{attribute 'OPC.UA.DA' :='1'}
	popa_0081_pt_3241_low_low_setpoint : REAL;
	//Alarm enable
	{attribute 'OPC.UA.DA' :='1'}
	popa_0081_pt_3241_low_low_enable: BOOL;
	
	//Alarm Priority setpoint
	{attribute 'OPC.UA.DA' :='1'}
	popa_0081_pt_3241_low_priority : INT;
	//Alarm delay setpoint(seconds)
	{attribute 'OPC.UA.DA' :='1'}
	popa_0081_pt_3241_low_delay_setpoint : INT;
	//Alarm active for HMI
	{attribute 'OPC.UA.DA' :='1'}
	popa_0081_pt_3241_low_active : BOOL;
	//Analog Alarm Setpoint
	{attribute 'OPC.UA.DA' :='1'}
	popa_0081_pt_3241_low_setpoint : REAL;
	//Alarm enable
	{attribute 'OPC.UA.DA' :='1'}
	popa_0081_pt_3241_low_enable: BOOL;
	
	//Alarm Priority setpoint
	{attribute 'OPC.UA.DA' :='1'}
	popa_0081_pt_3241_high_priority : INT;
	//Alarm delay setpoint(seconds)
	{attribute 'OPC.UA.DA' :='1'}
	popa_0081_pt_3241_high_delay_setpoint : INT;
	//Alarm active for HMI
	{attribute 'OPC.UA.DA' :='1'}
	popa_0081_pt_3241_high_active : BOOL;
	//Analog Alarm Setpoint
	{attribute 'OPC.UA.DA' :='1'}
	popa_0081_pt_3241_high_setpoint : REAL;
	//Alarm enable
	{attribute 'OPC.UA.DA' :='1'}
	popa_0081_pt_3241_high_enable: BOOL;
	
	//Alarm Priority setpoint
	{attribute 'OPC.UA.DA' :='1'}
	popa_0081_pt_3241_high_high_priority : INT;
	//Alarm delay setpoint(seconds)
	{attribute 'OPC.UA.DA' :='1'}
	popa_0081_pt_3241_high_high_delay_setpoint : INT;
	//Alarm active for HMI
	{attribute 'OPC.UA.DA' :='1'}
	popa_0081_pt_3241_high_high_active : BOOL;
	//Analog Alarm Setpoint
	{attribute 'OPC.UA.DA' :='1'}
	popa_0081_pt_3241_high_high_setpoint : REAL;
	//Alarm enable
	{attribute 'OPC.UA.DA' :='1'}
	popa_0081_pt_3241_high_high_enable: BOOL;
	
	
	//Raw Min value for analog input
	{attribute 'OPC.UA.DA' :='1'}
	popa_0081_pt_3241_raw_min : REAL :=0;
	//Raw max value for analog input
	{attribute 'OPC.UA.DA' :='1'}
	popa_0081_pt_3241_raw_max : REAL :=32767;
	//EU Min value for analog input
	{attribute 'OPC.UA.DA' :='1'}
	popa_0081_pt_3241_eu_min : REAL;
	//EU Max value for analog input
	{attribute 'OPC.UA.DA' :='1'}
	popa_0081_pt_3241_eu_max : REAL;
	//Filter factor value for analog input
	{attribute 'OPC.UA.DA' :='1'}
	popa_0081_pt_3241_filter_factor : REAL;
	//Scaled value for analog input
	{attribute 'OPC.UA.DA' :='1'}
	popa_0081_pt_3241_scaled_value : REAL;
	
	//---pt_3341-----------------------------------------------------------------------------------------------------------------------
	//Alarm Priority setpoint
	{attribute 'OPC.UA.DA' :='1'}
	popa_0081_pt_3341_low_low_priority : INT;
	//Alarm delay setpoint(seconds)
	{attribute 'OPC.UA.DA' :='1'}
	popa_0081_pt_3341_low_low_delay_setpoint : INT;
	//Alarm active for HMI
	{attribute 'OPC.UA.DA' :='1'}
	popa_0081_pt_3341_low_low_active : BOOL;
	//Analog Alarm Setpoint
	{attribute 'OPC.UA.DA' :='1'}
	popa_0081_pt_3341_low_low_setpoint : REAL;
	//Alarm enable
	{attribute 'OPC.UA.DA' :='1'}
	popa_0081_pt_3341_low_low_enable: BOOL;
	
	//Alarm Priority setpoint
	{attribute 'OPC.UA.DA' :='1'}
	popa_0081_pt_3341_low_priority : INT;
	//Alarm delay setpoint(seconds)
	{attribute 'OPC.UA.DA' :='1'}
	popa_0081_pt_3341_low_delay_setpoint : INT;
	//Alarm active for HMI
	{attribute 'OPC.UA.DA' :='1'}
	popa_0081_pt_3341_low_active : BOOL;
	//Analog Alarm Setpoint
	{attribute 'OPC.UA.DA' :='1'}
	popa_0081_pt_3341_low_setpoint : REAL;
	//Alarm enable
	{attribute 'OPC.UA.DA' :='1'}
	popa_0081_pt_3341_low_enable: BOOL;
	
	//Alarm Priority setpoint
	{attribute 'OPC.UA.DA' :='1'}
	popa_0081_pt_3341_high_priority : INT;
	//Alarm delay setpoint(seconds)
	{attribute 'OPC.UA.DA' :='1'}
	popa_0081_pt_3341_high_delay_setpoint : INT;
	//Alarm active for HMI
	{attribute 'OPC.UA.DA' :='1'}
	popa_0081_pt_3341_high_active : BOOL;
	//Analog Alarm Setpoint
	{attribute 'OPC.UA.DA' :='1'}
	popa_0081_pt_3341_high_setpoint : REAL;
	//Alarm enable
	{attribute 'OPC.UA.DA' :='1'}
	popa_0081_pt_3341_high_enable: BOOL;
	
	//Alarm Priority setpoint
	{attribute 'OPC.UA.DA' :='1'}
	popa_0081_pt_3341_high_high_priority : INT;
	//Alarm delay setpoint(seconds)
	{attribute 'OPC.UA.DA' :='1'}
	popa_0081_pt_3341_high_high_delay_setpoint : INT;
	//Alarm active for HMI
	{attribute 'OPC.UA.DA' :='1'}
	popa_0081_pt_3341_high_high_active : BOOL;
	//Analog Alarm Setpoint
	{attribute 'OPC.UA.DA' :='1'}
	popa_0081_pt_3341_high_high_setpoint : REAL;
	//Alarm enable
	{attribute 'OPC.UA.DA' :='1'}
	popa_0081_pt_3341_high_high_enable: BOOL;
	
	
	//Raw Min value for analog input
	{attribute 'OPC.UA.DA' :='1'}
	popa_0081_pt_3341_raw_min : REAL :=0;
	//Raw max value for analog input
	{attribute 'OPC.UA.DA' :='1'}
	popa_0081_pt_3341_raw_max : REAL :=32767;
	//EU Min value for analog input
	{attribute 'OPC.UA.DA' :='1'}
	popa_0081_pt_3341_eu_min : REAL;
	//EU Max value for analog input
	{attribute 'OPC.UA.DA' :='1'}
	popa_0081_pt_3341_eu_max : REAL;
	//Filter factor value for analog input
	{attribute 'OPC.UA.DA' :='1'}
	popa_0081_pt_3341_filter_factor : REAL;
	//Scaled value for analog input
	{attribute 'OPC.UA.DA' :='1'}
	popa_0081_pt_3341_scaled_value : REAL;
	
	//---tt_3118-----------------------------------------------------------------------------------------------------------------------
	//Alarm Priority setpoint
	{attribute 'OPC.UA.DA' :='1'}
	popa_0081_tt_3118_low_low_priority : INT;
	//Alarm delay setpoint(seconds)
	{attribute 'OPC.UA.DA' :='1'}
	popa_0081_tt_3118_low_low_delay_setpoint : INT;
	//Alarm active for HMI
	{attribute 'OPC.UA.DA' :='1'}
	popa_0081_tt_3118_low_low_active : BOOL;
	//Analog Alarm Setpoint
	{attribute 'OPC.UA.DA' :='1'}
	popa_0081_tt_3118_low_low_setpoint : REAL;
	//Alarm enable
	{attribute 'OPC.UA.DA' :='1'}
	popa_0081_tt_3118_low_low_enable: BOOL;
	
	//Alarm Priority setpoint
	{attribute 'OPC.UA.DA' :='1'}
	popa_0081_tt_3118_low_priority : INT;
	//Alarm delay setpoint(seconds)
	{attribute 'OPC.UA.DA' :='1'}
	popa_0081_tt_3118_low_delay_setpoint : INT;
	//Alarm active for HMI
	{attribute 'OPC.UA.DA' :='1'}
	popa_0081_tt_3118_low_active : BOOL;
	//Analog Alarm Setpoint
	{attribute 'OPC.UA.DA' :='1'}
	popa_0081_tt_3118_low_setpoint : REAL;
	//Alarm enable
	{attribute 'OPC.UA.DA' :='1'}
	popa_0081_tt_3118_low_enable: BOOL;
	
	//Alarm Priority setpoint
	{attribute 'OPC.UA.DA' :='1'}
	popa_0081_tt_3118_high_priority : INT;
	//Alarm delay setpoint(seconds)
	{attribute 'OPC.UA.DA' :='1'}
	popa_0081_tt_3118_high_delay_setpoint : INT;
	//Alarm active for HMI
	{attribute 'OPC.UA.DA' :='1'}
	popa_0081_tt_3118_high_active : BOOL;
	//Analog Alarm Setpoint
	{attribute 'OPC.UA.DA' :='1'}
	popa_0081_tt_3118_high_setpoint : REAL;
	//Alarm enable
	{attribute 'OPC.UA.DA' :='1'}
	popa_0081_tt_3118_high_enable: BOOL;
	
	//Alarm Priority setpoint
	{attribute 'OPC.UA.DA' :='1'}
	popa_0081_tt_3118_high_high_priority : INT;
	//Alarm delay setpoint(seconds)
	{attribute 'OPC.UA.DA' :='1'}
	popa_0081_tt_3118_high_high_delay_setpoint : INT;
	//Alarm active for HMI
	{attribute 'OPC.UA.DA' :='1'}
	popa_0081_tt_3118_high_high_active : BOOL;
	//Analog Alarm Setpoint
	{attribute 'OPC.UA.DA' :='1'}
	popa_0081_tt_3118_high_high_setpoint : REAL;
	//Alarm enable
	{attribute 'OPC.UA.DA' :='1'}
	popa_0081_tt_3118_high_high_enable: BOOL;
	
	
	//Raw Min value for analog input
	{attribute 'OPC.UA.DA' :='1'}
	popa_0081_tt_3118_raw_min : REAL :=0;
	//Raw max value for analog input
	{attribute 'OPC.UA.DA' :='1'}
	popa_0081_tt_3118_raw_max : REAL :=32767;
	//EU Min value for analog input
	{attribute 'OPC.UA.DA' :='1'}
	popa_0081_tt_3118_eu_min : REAL;
	//EU Max value for analog input
	{attribute 'OPC.UA.DA' :='1'}
	popa_0081_tt_3118_eu_max : REAL;
	//Filter factor value for analog input
	{attribute 'OPC.UA.DA' :='1'}
	popa_0081_tt_3118_filter_factor : REAL;
	//Scaled value for analog input
	{attribute 'OPC.UA.DA' :='1'}
	popa_0081_tt_3118_scaled_value : REAL;
	
	//---tt_3218-----------------------------------------------------------------------------------------------------------------------
	//Alarm Priority setpoint
	{attribute 'OPC.UA.DA' :='1'}
	popa_0081_tt_3218_low_low_priority : INT;
	//Alarm delay setpoint(seconds)
	{attribute 'OPC.UA.DA' :='1'}
	popa_0081_tt_3218_low_low_delay_setpoint : INT;
	//Alarm active for HMI
	{attribute 'OPC.UA.DA' :='1'}
	popa_0081_tt_3218_low_low_active : BOOL;
	//Analog Alarm Setpoint
	{attribute 'OPC.UA.DA' :='1'}
	popa_0081_tt_3218_low_low_setpoint : REAL;
	//Alarm enable
	{attribute 'OPC.UA.DA' :='1'}
	popa_0081_tt_3218_low_low_enable: BOOL;
	
	//Alarm Priority setpoint
	{attribute 'OPC.UA.DA' :='1'}
	popa_0081_tt_3218_low_priority : INT;
	//Alarm delay setpoint(seconds)
	{attribute 'OPC.UA.DA' :='1'}
	popa_0081_tt_3218_low_delay_setpoint : INT;
	//Alarm active for HMI
	{attribute 'OPC.UA.DA' :='1'}
	popa_0081_tt_3218_low_active : BOOL;
	//Analog Alarm Setpoint
	{attribute 'OPC.UA.DA' :='1'}
	popa_0081_tt_3218_low_setpoint : REAL;
	//Alarm enable
	{attribute 'OPC.UA.DA' :='1'}
	popa_0081_tt_3218_low_enable: BOOL;
	
	//Alarm Priority setpoint
	{attribute 'OPC.UA.DA' :='1'}
	popa_0081_tt_3218_high_priority : INT;
	//Alarm delay setpoint(seconds)
	{attribute 'OPC.UA.DA' :='1'}
	popa_0081_tt_3218_high_delay_setpoint : INT;
	//Alarm active for HMI
	{attribute 'OPC.UA.DA' :='1'}
	popa_0081_tt_3218_high_active : BOOL;
	//Analog Alarm Setpoint
	{attribute 'OPC.UA.DA' :='1'}
	popa_0081_tt_3218_high_setpoint : REAL;
	//Alarm enable
	{attribute 'OPC.UA.DA' :='1'}
	popa_0081_tt_3218_high_enable: BOOL;
	
	//Alarm Priority setpoint
	{attribute 'OPC.UA.DA' :='1'}
	popa_0081_tt_3218_high_high_priority : INT;
	//Alarm delay setpoint(seconds)
	{attribute 'OPC.UA.DA' :='1'}
	popa_0081_tt_3218_high_high_delay_setpoint : INT;
	//Alarm active for HMI
	{attribute 'OPC.UA.DA' :='1'}
	popa_0081_tt_3218_high_high_active : BOOL;
	//Analog Alarm Setpoint
	{attribute 'OPC.UA.DA' :='1'}
	popa_0081_tt_3218_high_high_setpoint : REAL;
	//Alarm enable
	{attribute 'OPC.UA.DA' :='1'}
	popa_0081_tt_3218_high_high_enable: BOOL;
	
	
	//Raw Min value for analog input
	{attribute 'OPC.UA.DA' :='1'}
	popa_0081_tt_3218_raw_min : REAL :=0;
	//Raw max value for analog input
	{attribute 'OPC.UA.DA' :='1'}
	popa_0081_tt_3218_raw_max : REAL :=32767;
	//EU Min value for analog input
	{attribute 'OPC.UA.DA' :='1'}
	popa_0081_tt_3218_eu_min : REAL;
	//EU Max value for analog input
	{attribute 'OPC.UA.DA' :='1'}
	popa_0081_tt_3218_eu_max : REAL;
	//Filter factor value for analog input
	{attribute 'OPC.UA.DA' :='1'}
	popa_0081_tt_3218_filter_factor : REAL;
	//Scaled value for analog input
	{attribute 'OPC.UA.DA' :='1'}
	popa_0081_tt_3218_scaled_value : REAL;
	
	//---tt_3318-----------------------------------------------------------------------------------------------------------------------
	//Alarm Priority setpoint
	{attribute 'OPC.UA.DA' :='1'}
	popa_0081_tt_3318_low_low_priority : INT;
	//Alarm delay setpoint(seconds)
	{attribute 'OPC.UA.DA' :='1'}
	popa_0081_tt_3318_low_low_delay_setpoint : INT;
	//Alarm active for HMI
	{attribute 'OPC.UA.DA' :='1'}
	popa_0081_tt_3318_low_low_active : BOOL;
	//Analog Alarm Setpoint
	{attribute 'OPC.UA.DA' :='1'}
	popa_0081_tt_3318_low_low_setpoint : REAL;
	//Alarm enable
	{attribute 'OPC.UA.DA' :='1'}
	popa_0081_tt_3318_low_low_enable: BOOL;
	
	//Alarm Priority setpoint
	{attribute 'OPC.UA.DA' :='1'}
	popa_0081_tt_3318_low_priority : INT;
	//Alarm delay setpoint(seconds)
	{attribute 'OPC.UA.DA' :='1'}
	popa_0081_tt_3318_low_delay_setpoint : INT;
	//Alarm active for HMI
	{attribute 'OPC.UA.DA' :='1'}
	popa_0081_tt_3318_low_active : BOOL;
	//Analog Alarm Setpoint
	{attribute 'OPC.UA.DA' :='1'}
	popa_0081_tt_3318_low_setpoint : REAL;
	//Alarm enable
	{attribute 'OPC.UA.DA' :='1'}
	popa_0081_tt_3318_low_enable: BOOL;
	
	//Alarm Priority setpoint
	{attribute 'OPC.UA.DA' :='1'}
	popa_0081_tt_3318_high_priority : INT;
	//Alarm delay setpoint(seconds)
	{attribute 'OPC.UA.DA' :='1'}
	popa_0081_tt_3318_high_delay_setpoint : INT;
	//Alarm active for HMI
	{attribute 'OPC.UA.DA' :='1'}
	popa_0081_tt_3318_high_active : BOOL;
	//Analog Alarm Setpoint
	{attribute 'OPC.UA.DA' :='1'}
	popa_0081_tt_3318_high_setpoint : REAL;
	//Alarm enable
	{attribute 'OPC.UA.DA' :='1'}
	popa_0081_tt_3318_high_enable: BOOL;
	
	//Alarm Priority setpoint
	{attribute 'OPC.UA.DA' :='1'}
	popa_0081_tt_3318_high_high_priority : INT;
	//Alarm delay setpoint(seconds)
	{attribute 'OPC.UA.DA' :='1'}
	popa_0081_tt_3318_high_high_delay_setpoint : INT;
	//Alarm active for HMI
	{attribute 'OPC.UA.DA' :='1'}
	popa_0081_tt_3318_high_high_active : BOOL;
	//Analog Alarm Setpoint
	{attribute 'OPC.UA.DA' :='1'}
	popa_0081_tt_3318_high_high_setpoint : REAL;
	//Alarm enable
	{attribute 'OPC.UA.DA' :='1'}
	popa_0081_tt_3318_high_high_enable: BOOL;
	
	
	//Raw Min value for analog input
	{attribute 'OPC.UA.DA' :='1'}
	popa_0081_tt_3318_raw_min : REAL :=0;
	//Raw max value for analog input
	{attribute 'OPC.UA.DA' :='1'}
	popa_0081_tt_3318_raw_max : REAL :=32767;
	//EU Min value for analog input
	{attribute 'OPC.UA.DA' :='1'}
	popa_0081_tt_3318_eu_min : REAL;
	//EU Max value for analog input
	{attribute 'OPC.UA.DA' :='1'}
	popa_0081_tt_3318_eu_max : REAL;
	//Filter factor value for analog input
	{attribute 'OPC.UA.DA' :='1'}
	popa_0081_tt_3318_filter_factor : REAL;
	//Scaled value for analog input
	{attribute 'OPC.UA.DA' :='1'}
	popa_0081_tt_3318_scaled_value : REAL;
	
	//---tt_3140-----------------------------------------------------------------------------------------------------------------------
	//Alarm Priority setpoint
	{attribute 'OPC.UA.DA' :='1'}
	popa_0081_tt_3140_low_low_priority : INT;
	//Alarm delay setpoint(seconds)
	{attribute 'OPC.UA.DA' :='1'}
	popa_0081_tt_3140_low_low_delay_setpoint : INT;
	//Alarm active for HMI
	{attribute 'OPC.UA.DA' :='1'}
	popa_0081_tt_3140_low_low_active : BOOL;
	//Analog Alarm Setpoint
	{attribute 'OPC.UA.DA' :='1'}
	popa_0081_tt_3140_low_low_setpoint : REAL;
	//Alarm enable
	{attribute 'OPC.UA.DA' :='1'}
	popa_0081_tt_3140_low_low_enable: BOOL;
	
	//Alarm Priority setpoint
	{attribute 'OPC.UA.DA' :='1'}
	popa_0081_tt_3140_low_priority : INT;
	//Alarm delay setpoint(seconds)
	{attribute 'OPC.UA.DA' :='1'}
	popa_0081_tt_3140_low_delay_setpoint : INT;
	//Alarm active for HMI
	{attribute 'OPC.UA.DA' :='1'}
	popa_0081_tt_3140_low_active : BOOL;
	//Analog Alarm Setpoint
	{attribute 'OPC.UA.DA' :='1'}
	popa_0081_tt_3140_low_setpoint : REAL;
	//Alarm enable
	{attribute 'OPC.UA.DA' :='1'}
	popa_0081_tt_3140_low_enable: BOOL;
	
	//Alarm Priority setpoint
	{attribute 'OPC.UA.DA' :='1'}
	popa_0081_tt_3140_high_priority : INT;
	//Alarm delay setpoint(seconds)
	{attribute 'OPC.UA.DA' :='1'}
	popa_0081_tt_3140_high_delay_setpoint : INT;
	//Alarm active for HMI
	{attribute 'OPC.UA.DA' :='1'}
	popa_0081_tt_3140_high_active : BOOL;
	//Analog Alarm Setpoint
	{attribute 'OPC.UA.DA' :='1'}
	popa_0081_tt_3140_high_setpoint : REAL;
	//Alarm enable
	{attribute 'OPC.UA.DA' :='1'}
	popa_0081_tt_3140_high_enable: BOOL;
	
	//Alarm Priority setpoint
	{attribute 'OPC.UA.DA' :='1'}
	popa_0081_tt_3140_high_high_priority : INT;
	//Alarm delay setpoint(seconds)
	{attribute 'OPC.UA.DA' :='1'}
	popa_0081_tt_3140_high_high_delay_setpoint : INT;
	//Alarm active for HMI
	{attribute 'OPC.UA.DA' :='1'}
	popa_0081_tt_3140_high_high_active : BOOL;
	//Analog Alarm Setpoint
	{attribute 'OPC.UA.DA' :='1'}
	popa_0081_tt_3140_high_high_setpoint : REAL;
	//Alarm enable
	{attribute 'OPC.UA.DA' :='1'}
	popa_0081_tt_3140_high_high_enable: BOOL;
	
	
	//Raw Min value for analog input
	{attribute 'OPC.UA.DA' :='1'}
	popa_0081_tt_3140_raw_min : REAL :=0;
	//Raw max value for analog input
	{attribute 'OPC.UA.DA' :='1'}
	popa_0081_tt_3140_raw_max : REAL :=32767;
	//EU Min value for analog input
	{attribute 'OPC.UA.DA' :='1'}
	popa_0081_tt_3140_eu_min : REAL;
	//EU Max value for analog input
	{attribute 'OPC.UA.DA' :='1'}
	popa_0081_tt_3140_eu_max : REAL;
	//Filter factor value for analog input
	{attribute 'OPC.UA.DA' :='1'}
	popa_0081_tt_3140_filter_factor : REAL;
	//Scaled value for analog input
	{attribute 'OPC.UA.DA' :='1'}
	popa_0081_tt_3140_scaled_value : REAL;
	
	//---tt_3240-----------------------------------------------------------------------------------------------------------------------
	//Alarm Priority setpoint
	{attribute 'OPC.UA.DA' :='1'}
	popa_0081_tt_3240_low_low_priority : INT;
	//Alarm delay setpoint(seconds)
	{attribute 'OPC.UA.DA' :='1'}
	popa_0081_tt_3240_low_low_delay_setpoint : INT;
	//Alarm active for HMI
	{attribute 'OPC.UA.DA' :='1'}
	popa_0081_tt_3240_low_low_active : BOOL;
	//Analog Alarm Setpoint
	{attribute 'OPC.UA.DA' :='1'}
	popa_0081_tt_3240_low_low_setpoint : REAL;
	//Alarm enable
	{attribute 'OPC.UA.DA' :='1'}
	popa_0081_tt_3240_low_low_enable: BOOL;
	
	//Alarm Priority setpoint
	{attribute 'OPC.UA.DA' :='1'}
	popa_0081_tt_3240_low_priority : INT;
	//Alarm delay setpoint(seconds)
	{attribute 'OPC.UA.DA' :='1'}
	popa_0081_tt_3240_low_delay_setpoint : INT;
	//Alarm active for HMI
	{attribute 'OPC.UA.DA' :='1'}
	popa_0081_tt_3240_low_active : BOOL;
	//Analog Alarm Setpoint
	{attribute 'OPC.UA.DA' :='1'}
	popa_0081_tt_3240_low_setpoint : REAL;
	//Alarm enable
	{attribute 'OPC.UA.DA' :='1'}
	popa_0081_tt_3240_low_enable: BOOL;
	
	//Alarm Priority setpoint
	{attribute 'OPC.UA.DA' :='1'}
	popa_0081_tt_3240_high_priority : INT;
	//Alarm delay setpoint(seconds)
	{attribute 'OPC.UA.DA' :='1'}
	popa_0081_tt_3240_high_delay_setpoint : INT;
	//Alarm active for HMI
	{attribute 'OPC.UA.DA' :='1'}
	popa_0081_tt_3240_high_active : BOOL;
	//Analog Alarm Setpoint
	{attribute 'OPC.UA.DA' :='1'}
	popa_0081_tt_3240_high_setpoint : REAL;
	//Alarm enable
	{attribute 'OPC.UA.DA' :='1'}
	popa_0081_tt_3240_high_enable: BOOL;
	
	//Alarm Priority setpoint
	{attribute 'OPC.UA.DA' :='1'}
	popa_0081_tt_3240_high_high_priority : INT;
	//Alarm delay setpoint(seconds)
	{attribute 'OPC.UA.DA' :='1'}
	popa_0081_tt_3240_high_high_delay_setpoint : INT;
	//Alarm active for HMI
	{attribute 'OPC.UA.DA' :='1'}
	popa_0081_tt_3240_high_high_active : BOOL;
	//Analog Alarm Setpoint
	{attribute 'OPC.UA.DA' :='1'}
	popa_0081_tt_3240_high_high_setpoint : REAL;
	//Alarm enable
	{attribute 'OPC.UA.DA' :='1'}
	popa_0081_tt_3240_high_high_enable: BOOL;
	
	
	//Raw Min value for analog input
	{attribute 'OPC.UA.DA' :='1'}
	popa_0081_tt_3240_raw_min : REAL :=0;
	//Raw max value for analog input
	{attribute 'OPC.UA.DA' :='1'}
	popa_0081_tt_3240_raw_max : REAL :=32767;
	//EU Min value for analog input
	{attribute 'OPC.UA.DA' :='1'}
	popa_0081_tt_3240_eu_min : REAL;
	//EU Max value for analog input
	{attribute 'OPC.UA.DA' :='1'}
	popa_0081_tt_3240_eu_max : REAL;
	//Filter factor value for analog input
	{attribute 'OPC.UA.DA' :='1'}
	popa_0081_tt_3240_filter_factor : REAL;
	//Scaled value for analog input
	{attribute 'OPC.UA.DA' :='1'}
	popa_0081_tt_3240_scaled_value : REAL;
	
	//---tt_3340-----------------------------------------------------------------------------------------------------------------------
	//Alarm Priority setpoint
	{attribute 'OPC.UA.DA' :='1'}
	popa_0081_tt_3340_low_low_priority : INT;
	//Alarm delay setpoint(seconds)
	{attribute 'OPC.UA.DA' :='1'}
	popa_0081_tt_3340_low_low_delay_setpoint : INT;
	//Alarm active for HMI
	{attribute 'OPC.UA.DA' :='1'}
	popa_0081_tt_3340_low_low_active : BOOL;
	//Analog Alarm Setpoint
	{attribute 'OPC.UA.DA' :='1'}
	popa_0081_tt_3340_low_low_setpoint : REAL;
	//Alarm enable
	{attribute 'OPC.UA.DA' :='1'}
	popa_0081_tt_3340_low_low_enable: BOOL;
	
	//Alarm Priority setpoint
	{attribute 'OPC.UA.DA' :='1'}
	popa_0081_tt_3340_low_priority : INT;
	//Alarm delay setpoint(seconds)
	{attribute 'OPC.UA.DA' :='1'}
	popa_0081_tt_3340_low_delay_setpoint : INT;
	//Alarm active for HMI
	{attribute 'OPC.UA.DA' :='1'}
	popa_0081_tt_3340_low_active : BOOL;
	//Analog Alarm Setpoint
	{attribute 'OPC.UA.DA' :='1'}
	popa_0081_tt_3340_low_setpoint : REAL;
	//Alarm enable
	{attribute 'OPC.UA.DA' :='1'}
	popa_0081_tt_3340_low_enable: BOOL;
	
	//Alarm Priority setpoint
	{attribute 'OPC.UA.DA' :='1'}
	popa_0081_tt_3340_high_priority : INT;
	//Alarm delay setpoint(seconds)
	{attribute 'OPC.UA.DA' :='1'}
	popa_0081_tt_3340_high_delay_setpoint : INT;
	//Alarm active for HMI
	{attribute 'OPC.UA.DA' :='1'}
	popa_0081_tt_3340_high_active : BOOL;
	//Analog Alarm Setpoint
	{attribute 'OPC.UA.DA' :='1'}
	popa_0081_tt_3340_high_setpoint : REAL;
	//Alarm enable
	{attribute 'OPC.UA.DA' :='1'}
	popa_0081_tt_3340_high_enable: BOOL;
	
	//Alarm Priority setpoint
	{attribute 'OPC.UA.DA' :='1'}
	popa_0081_tt_3340_high_high_priority : INT;
	//Alarm delay setpoint(seconds)
	{attribute 'OPC.UA.DA' :='1'}
	popa_0081_tt_3340_high_high_delay_setpoint : INT;
	//Alarm active for HMI
	{attribute 'OPC.UA.DA' :='1'}
	popa_0081_tt_3340_high_high_active : BOOL;
	//Analog Alarm Setpoint
	{attribute 'OPC.UA.DA' :='1'}
	popa_0081_tt_3340_high_high_setpoint : REAL;
	//Alarm enable
	{attribute 'OPC.UA.DA' :='1'}
	popa_0081_tt_3340_high_high_enable: BOOL;
	
	
	//Raw Min value for analog input
	{attribute 'OPC.UA.DA' :='1'}
	popa_0081_tt_3340_raw_min : REAL :=0;
	//Raw max value for analog input
	{attribute 'OPC.UA.DA' :='1'}
	popa_0081_tt_3340_raw_max : REAL :=32767;
	//EU Min value for analog input
	{attribute 'OPC.UA.DA' :='1'}
	popa_0081_tt_3340_eu_min : REAL;
	//EU Max value for analog input
	{attribute 'OPC.UA.DA' :='1'}
	popa_0081_tt_3340_eu_max : REAL;
	//Filter factor value for analog input
	{attribute 'OPC.UA.DA' :='1'}
	popa_0081_tt_3340_filter_factor : REAL;
	//Scaled value for analog input
	{attribute 'OPC.UA.DA' :='1'}
	popa_0081_tt_3340_scaled_value : REAL;
	
END_VAR

(* stored: Version 1.1.0.1, ProductVersion 3.1.4024.12
   GVL opc: Id {674fd3be-a48d-4a85-a2e2-bd0824412020} *)
